   1:  PR[GP1:91,2] = PR[GP1:90,2] + 99.468;
   1:L PR[91] 10mm/sec FINE;
   1:  PR[GP1:91,1] = PR[GP1:90,1] + 74.034;
   1:  PR[GP1:91,2] = PR[GP1:90,2] + 97.039;
   1:L PR[91] 10mm/sec FINE;
   1:  PR[GP1:91,1] = PR[GP1:90,1] + 75.968;
   1:  PR[GP1:91,2] = PR[GP1:90,2] + 94.856;
   1:L PR[91] 10mm/sec FINE;
   1:  PR[GP1:91,1] = PR[GP1:90,1] + 77.516;
   1:  PR[GP1:91,2] = PR[GP1:90,2] + 93.858;
   1:  PR[GP1:91,3] = PR[GP1:90,3] + 42.900;
   1:L PR[91] 10mm/sec FINE;
   1:  PR[GP1:91,1] = PR[GP1:90,1] + 79.283;
   1:  PR[GP1:91,2] = PR[GP1:90,2] + 92.339;
   1:L PR[91] 10mm/sec FINE;
   1:  PR[GP1:91,1] = PR[GP1:90,1] + 81.543;
   1:  PR[GP1:91,2] = PR[GP1:90,2] + 90.798;
   1:L PR[91] 10mm/sec FINE;
   1:  PR[GP1:91,1] = PR[GP1:90,1] + 82.942;
   1:  PR[GP1:91,2] = PR[GP1:90,2] + 89.888;
   1:L PR[91] 10mm/sec FINE;
   1:  PR[GP1:91,1] = PR[GP1:90,1] + 83.980;
   1:  PR[GP1:91,2] = PR[GP1:90,2] + 89.382;
   1:L PR[91] 10mm/sec FINE;
   1:  PR[GP1:91,1] = PR[GP1:90,1] + 87.933;
   1:  PR[GP1:91,2] = PR[GP1:90,2] + 87.648;
   1:L PR[91] 10mm/sec FINE;
   1:  PR[GP1:91,1] = PR[GP1:90,1] + 88.187;
   1:  PR[GP1:91,2] = PR[GP1:90,2] + 87.560;
   1:L PR[91] 10mm/sec FINE;
   1:  PR[GP1:91,1] = PR[GP1:90,1] + 89.431;
   1:  PR[GP1:91,2] = PR[GP1:90,2] + 87.262;
   1:L PR[91] 10mm/sec FINE;
   1:  PR[GP1:91,1] = PR[GP1:90,1] + 92.833;
   1:  PR[GP1:91,2] = PR[GP1:90,2] + 86.250;
   1:L PR[91] 10mm/sec FINE;
   1:  PR[GP1:91,1] = PR[GP1:90,1] + 93.950;
   1:  PR[GP1:91,2] = PR[GP1:90,2] + 85.987;
   1:L PR[91] 10mm/sec FINE;
   1:  PR[GP1:91,1] = PR[GP1:90,1] + 97.467;
   1:  PR[GP1:91,2] = PR[GP1:90,2] + 85.608;
   1:L PR[91] 10mm/sec FINE;
   1:  PR[GP1:91,1] = PR[GP1:90,1] + 100.046;
   1:  PR[GP1:91,2] = PR[GP1:90,2] + 85.501;
   1:L PR[91] 10mm/sec FINE;
   1:  PR[GP1:91,1] = PR[GP1:90,1] + 101.809;
   1:  PR[GP1:91,2] = PR[GP1:90,2] + 85.697;
   1:L PR[91] 10mm/sec FINE;
   1:  PR[GP1:91,1] = PR[GP1:90,1] + 102.507;
   1:  PR[GP1:91,2] = PR[GP1:90,2] + 85.656;
   1:L PR[91] 10mm/sec FINE;
   1:  PR[GP1:91,1] = PR[GP1:90,1] + 104.081;
   1:  PR[GP1:91,2] = PR[GP1:90,2] + 85.414;
   1:L PR[91] 10mm/sec FINE;
   1:  PR[GP1:91,1] = PR[GP1:90,1] + 105.629;
   1:  PR[GP1:91,2] = PR[GP1:90,2] + 85.297;
   1:L PR[91] 10mm/sec FINE;
   1:  PR[GP1:91,1] = PR[GP1:90,1] + 106.776;
   1:L PR[91] 10mm/sec FINE;
   1:  PR[GP1:91,1] = PR[GP1:90,1] + 108.676;
   1:  PR[GP1:91,2] = PR[GP1:90,2] + 85.462;
   1:L PR[91] 10mm/sec FINE;
   1:  PR[GP1:91,1] = PR[GP1:90,1] + 109.474;
   1:  PR[GP1:91,2] = PR[GP1:90,2] + 85.591;
   1:L PR[91] 10mm/sec FINE;
   1:  PR[GP1:91,1] = PR[GP1:90,1] + 111.613;
   1:  PR[GP1:91,2] = PR[GP1:90,2] + 86.140;
   1:L PR[91] 10mm/sec FINE;
   1:  PR[GP1:91,1] = PR[GP1:90,1] + 112.123;
   1:  PR[GP1:91,2] = PR[GP1:90,2] + 86.310;
   1:L PR[91] 10mm/sec FINE;
   1:  PR[GP1:91,1] = PR[GP1:90,1] + 114.339;
   1:  PR[GP1:91,2] = PR[GP1:90,2] + 87.294;
   1:L PR[91] 10mm/sec FINE;
   1:  PR[GP1:91,1] = PR[GP1:90,1] + 114.659;
   1:  PR[GP1:91,2] = PR[GP1:90,2] + 87.463;
   1:L PR[91] 10mm/sec FINE;
   1:  PR[GP1:91,1] = PR[GP1:90,1] + 116.762;
   1:  PR[GP1:91,2] = PR[GP1:90,2] + 88.857;
   1:L PR[91] 10mm/sec FINE;
   1:  PR[GP1:91,1] = PR[GP1:90,1] + 117.014;
   1:  PR[GP1:91,2] = PR[GP1:90,2] + 89.048;
   1:L PR[91] 10mm/sec FINE;
   1:  PR[GP1:91,1] = PR[GP1:90,1] + 118.819;
   1:  PR[GP1:91,2] = PR[GP1:90,2] + 90.739;
   1:L PR[91] 10mm/sec FINE;
   1:  PR[GP1:91,1] = PR[GP1:90,1] + 119.110;
   1:  PR[GP1:91,2] = PR[GP1:90,2] + 91.046;
   1:L PR[91] 10mm/sec FINE;
   1:  PR[GP1:91,1] = PR[GP1:90,1] + 120.475;
   1:  PR[GP1:91,2] = PR[GP1:90,2] + 92.841;
   1:L PR[91] 10mm/sec FINE;
   1:  PR[GP1:91,1] = PR[GP1:90,1] + 120.865;
   1:  PR[GP1:91,2] = PR[GP1:90,2] + 93.418;
   1:L PR[91] 10mm/sec FINE;
   1:  PR[GP1:91,1] = PR[GP1:90,1] + 121.741;
   1:  PR[GP1:91,2] = PR[GP1:90,2] + 95.070;
   1:L PR[91] 10mm/sec FINE;
   1:  PR[GP1:91,1] = PR[GP1:90,1] + 122.220;
   1:  PR[GP1:91,2] = PR[GP1:90,2] + 96.089;
   1:L PR[91] 10mm/sec FINE;
   1:  PR[GP1:91,1] = PR[GP1:90,1] + 122.659;
   1:  PR[GP1:91,2] = PR[GP1:90,2] + 97.354;
   1:L PR[91] 10mm/sec FINE;
   1:  PR[GP1:91,1] = PR[GP1:90,1] + 123.139;
   1:  PR[GP1:91,2] = PR[GP1:90,2] + 98.958;
   1:L PR[91] 10mm/sec FINE;
   1:  PR[GP1:91,1] = PR[GP1:90,1] + 123.264;
   1:  PR[GP1:91,2] = PR[GP1:90,2] + 99.651;
   1:L PR[91] 10mm/sec FINE;
   1:  PR[GP1:91,1] = PR[GP1:90,1] + 123.588;
   1:  PR[GP1:91,2] = PR[GP1:90,2] + 101.921;
   1:L PR[91] 10mm/sec FINE;
   1:  PR[GP1:91,1] = PR[GP1:90,1] + 123.600;
   1:  PR[GP1:91,2] = PR[GP1:90,2] + 104.888;
   1:L PR[91] 10mm/sec FINE;
   1:  PR[GP1:91,1] = PR[GP1:90,1] + 122.995;
   1:  PR[GP1:91,2] = PR[GP1:90,2] + 108.791;
   1:L PR[91] 10mm/sec FINE;
   1:  PR[GP1:91,1] = PR[GP1:90,1] + 121.765;
   1:  PR[GP1:91,2] = PR[GP1:90,2] + 112.407;
   1:L PR[91] 10mm/sec FINE;
   1:  PR[GP1:91,1] = PR[GP1:90,1] + 120.870;
   1:  PR[GP1:91,2] = PR[GP1:90,2] + 113.981;
   1:L PR[91] 10mm/sec FINE;
   1:  PR[GP1:91,1] = PR[GP1:90,1] + 119.893;
   1:  PR[GP1:91,2] = PR[GP1:90,2] + 115.630;
   1:L PR[91] 10mm/sec FINE;
   1:  PR[GP1:91,1] = PR[GP1:90,1] + 119.147;
   1:  PR[GP1:91,2] = PR[GP1:90,2] + 116.492;
   1:L PR[91] 10mm/sec FINE;
   1:  PR[GP1:91,1] = PR[GP1:90,1] + 117.485;
   1:  PR[GP1:91,2] = PR[GP1:90,2] + 118.360;
   1:L PR[91] 10mm/sec FINE;
   1:  PR[GP1:91,1] = PR[GP1:90,1] + 114.657;
   1:  PR[GP1:91,2] = PR[GP1:90,2] + 120.517;
   1:L PR[91] 10mm/sec FINE;
   1:  PR[GP1:91,1] = PR[GP1:90,1] + 111.519;
   1:  PR[GP1:91,2] = PR[GP1:90,2] + 122.048;
   1:L PR[91] 10mm/sec FINE;
   1:  PR[GP1:91,1] = PR[GP1:90,1] + 110.087;
   1:  PR[GP1:91,2] = PR[GP1:90,2] + 122.431;
   1:L PR[91] 10mm/sec FINE;
   1:  PR[GP1:91,1] = PR[GP1:90,1] + 108.168;
   1:  PR[GP1:91,2] = PR[GP1:90,2] + 122.921;
   1:L PR[91] 10mm/sec FINE;
   1:  PR[GP1:91,1] = PR[GP1:90,1] + 104.699;
   1:  PR[GP1:91,2] = PR[GP1:90,2] + 123.124;
   1:L PR[91] 10mm/sec FINE;
   1:  PR[GP1:91,1] = PR[GP1:90,1] + 103.027;
   1:  PR[GP1:91,2] = PR[GP1:90,2] + 122.912;
   1:L PR[91] 10mm/sec FINE;
   1:  PR[GP1:91,1] = PR[GP1:90,1] + 101.276;
   1:  PR[GP1:91,2] = PR[GP1:90,2] + 122.649;
   1:L PR[91] 10mm/sec FINE;
   1:  PR[GP1:91,1] = PR[GP1:90,1] + 99.074;
   1:  PR[GP1:91,2] = PR[GP1:90,2] + 122.005;
   1:L PR[91] 10mm/sec FINE;
   1:  PR[GP1:91,1] = PR[GP1:90,1] + 97.904;
   1:  PR[GP1:91,2] = PR[GP1:90,2] + 121.902;
   1:L PR[91] 10mm/sec FINE;
   1:  PR[GP1:91,1] = PR[GP1:90,1] + 93.801;
   1:  PR[GP1:91,2] = PR[GP1:90,2] + 122.579;
   1:L PR[91] 10mm/sec FINE;
   1:  PR[GP1:91,1] = PR[GP1:90,1] + 93.286;
   1:  PR[GP1:91,2] = PR[GP1:90,2] + 122.645;
   1:L PR[91] 10mm/sec FINE;
   1:  PR[GP1:91,1] = PR[GP1:90,1] + 89.093;
   1:  PR[GP1:91,2] = PR[GP1:90,2] + 122.677;
   1:L PR[91] 10mm/sec FINE;
   1:  PR[GP1:91,1] = PR[GP1:90,1] + 87.629;
   1:  PR[GP1:91,2] = PR[GP1:90,2] + 122.537;
   1:L PR[91] 10mm/sec FINE;
   1:  PR[GP1:91,1] = PR[GP1:90,1] + 85.652;
   1:  PR[GP1:91,2] = PR[GP1:90,2] + 122.207;
   1:L PR[91] 10mm/sec FINE;
   1:  PR[GP1:91,1] = PR[GP1:90,1] + 83.813;
   1:  PR[GP1:91,2] = PR[GP1:90,2] + 121.808;
   1:L PR[91] 10mm/sec FINE;
   1:  PR[GP1:91,1] = PR[GP1:90,1] + 80.795;
   1:  PR[GP1:91,2] = PR[GP1:90,2] + 120.737;
   1:L PR[91] 10mm/sec FINE;
   1:  PR[GP1:91,1] = PR[GP1:90,1] + 78.461;
   1:  PR[GP1:91,2] = PR[GP1:90,2] + 119.530;
   1:L PR[91] 10mm/sec FINE;
   1:  PR[GP1:91,1] = PR[GP1:90,1] + 77.949;
   1:  PR[GP1:91,2] = PR[GP1:90,2] + 119.170;
   1:L PR[91] 10mm/sec FINE;
   1:  PR[GP1:91,1] = PR[GP1:90,1] + 76.319;
   1:  PR[GP1:91,2] = PR[GP1:90,2] + 117.935;
   1:L PR[91] 10mm/sec FINE;
   1:  PR[GP1:91,1] = PR[GP1:90,1] + 74.935;
   1:  PR[GP1:91,2] = PR[GP1:90,2] + 116.491;
   1:L PR[91] 10mm/sec FINE;
   1:  PR[GP1:91,1] = PR[GP1:90,1] + 74.408;
   1:  PR[GP1:91,2] = PR[GP1:90,2] + 115.908;
   1:L PR[91] 10mm/sec FINE;
   1:  PR[GP1:91,1] = PR[GP1:90,1] + 73.372;
   1:  PR[GP1:91,2] = PR[GP1:90,2] + 114.394;
   1:L PR[91] 10mm/sec FINE;
   1:  PR[GP1:91,1] = PR[GP1:90,1] + 72.842;
   1:  PR[GP1:91,2] = PR[GP1:90,2] + 113.448;
   1:L PR[91] 10mm/sec FINE;
   1:  PR[GP1:91,1] = PR[GP1:90,1] + 72.127;
   1:  PR[GP1:91,2] = PR[GP1:90,2] + 111.928;
   1:L PR[91] 10mm/sec FINE;
   1:  PR[GP1:91,1] = PR[GP1:90,1] + 71.355;
   1:  PR[GP1:91,2] = PR[GP1:90,2] + 109.313;
   1:L PR[91] 10mm/sec FINE;
   1:  PR[GP1:91,1] = PR[GP1:90,1] + 71.204;
   1:  PR[GP1:91,2] = PR[GP1:90,2] + 107.968;
   1:L PR[91] 10mm/sec FINE;
   1:  PR[GP1:91,1] = PR[GP1:90,1] + 71.186;
   1:  PR[GP1:91,2] = PR[GP1:90,2] + 106.809;
   1:L PR[91] 10mm/sec FINE;
   1:  PR[GP1:91,1] = PR[GP1:90,1] + 71.282;
   1:  PR[GP1:91,2] = PR[GP1:90,2] + 105.487;
   1:L PR[91] 10mm/sec FINE;
   1:  PR[GP1:91,1] = PR[GP1:90,1] + 71.483;
   1:  PR[GP1:91,2] = PR[GP1:90,2] + 104.578;
   1:L PR[91] 10mm/sec FINE;
   1:  PR[GP1:91,1] = PR[GP1:90,1] + 72.043;
   1:  PR[GP1:91,2] = PR[GP1:90,2] + 102.143;
   1:L PR[91] 10mm/sec FINE;
   1:  PR[GP1:91,1] = PR[GP1:90,1] + 73.160;
   1:  PR[GP1:91,2] = PR[GP1:90,2] + 99.391;
   1:L PR[91] 10mm/sec FINE;
   1:  PR[GP1:91,1] = PR[GP1:90,1] + 74.854;
   1:  PR[GP1:91,2] = PR[GP1:90,2] + 96.763;
   1:L PR[91] 10mm/sec FINE;
   1:  PR[GP1:91,1] = PR[GP1:90,1] + 76.583;
   1:  PR[GP1:91,2] = PR[GP1:90,2] + 94.811;
   1:L PR[91] 10mm/sec FINE;
   1:  PR[GP1:91,1] = PR[GP1:90,1] + 78.494;
   1:  PR[GP1:91,2] = PR[GP1:90,2] + 93.442;
   1:  PR[GP1:91,3] = PR[GP1:90,3] + 43.900;
   1:L PR[91] 10mm/sec FINE;
   1:  PR[GP1:91,1] = PR[GP1:90,1] + 79.972;
   1:  PR[GP1:91,2] = PR[GP1:90,2] + 92.171;
   1:L PR[91] 10mm/sec FINE;
   1:  PR[GP1:91,1] = PR[GP1:90,1] + 82.774;
   1:  PR[GP1:91,2] = PR[GP1:90,2] + 90.260;
   1:L PR[91] 10mm/sec FINE;
   1:  PR[GP1:91,1] = PR[GP1:90,1] + 83.771;
   1:  PR[GP1:91,2] = PR[GP1:90,2] + 89.611;
   1:L PR[91] 10mm/sec FINE;
   1:  PR[GP1:91,1] = PR[GP1:90,1] + 84.510;
   1:  PR[GP1:91,2] = PR[GP1:90,2] + 89.252;
   1:L PR[91] 10mm/sec FINE;
   1:  PR[GP1:91,1] = PR[GP1:90,1] + 88.374;
   1:  PR[GP1:91,2] = PR[GP1:90,2] + 87.556;
   1:L PR[91] 10mm/sec FINE;
   1:  PR[GP1:91,1] = PR[GP1:90,1] + 88.959;
   1:  PR[GP1:91,2] = PR[GP1:90,2] + 87.272;
   1:L PR[91] 10mm/sec FINE;
   1:  PR[GP1:91,1] = PR[GP1:90,1] + 93.314;
   1:  PR[GP1:91,2] = PR[GP1:90,2] + 85.976;
   1:L PR[91] 10mm/sec FINE;
   1:  PR[GP1:91,1] = PR[GP1:90,1] + 94.968;
   1:  PR[GP1:91,2] = PR[GP1:90,2] + 85.587;
   1:L PR[91] 10mm/sec FINE;
   1:  PR[GP1:91,1] = PR[GP1:90,1] + 97.962;
   1:  PR[GP1:91,2] = PR[GP1:90,2] + 85.265;
   1:L PR[91] 10mm/sec FINE;
   1:  PR[GP1:91,1] = PR[GP1:90,1] + 101.083;
   1:  PR[GP1:91,2] = PR[GP1:90,2] + 85.135;
   1:L PR[91] 10mm/sec FINE;
   1:  PR[GP1:91,1] = PR[GP1:90,1] + 102.373;
   1:  PR[GP1:91,2] = PR[GP1:90,2] + 85.288;
   1:L PR[91] 10mm/sec FINE;
   1:  PR[GP1:91,1] = PR[GP1:90,1] + 103.011;
   1:  PR[GP1:91,2] = PR[GP1:90,2] + 85.251;
   1:L PR[91] 10mm/sec FINE;
   1:  PR[GP1:91,1] = PR[GP1:90,1] + 103.965;
   1:  PR[GP1:91,2] = PR[GP1:90,2] + 85.105;
   1:L PR[91] 10mm/sec FINE;
   1:  PR[GP1:91,1] = PR[GP1:90,1] + 106.183;
   1:  PR[GP1:91,2] = PR[GP1:90,2] + 84.937;
   1:L PR[91] 10mm/sec FINE;
   1:  PR[GP1:91,1] = PR[GP1:90,1] + 106.658;
   1:L PR[91] 10mm/sec FINE;
   1:  PR[GP1:91,1] = PR[GP1:90,1] + 109.269;
   1:  PR[GP1:91,2] = PR[GP1:90,2] + 85.163;
   1:L PR[91] 10mm/sec FINE;
   1:  PR[GP1:91,1] = PR[GP1:90,1] + 112.218;
   1:  PR[GP1:91,2] = PR[GP1:90,2] + 85.893;
   1:L PR[91] 10mm/sec FINE;
   1:  PR[GP1:91,1] = PR[GP1:90,1] + 114.511;
   1:  PR[GP1:91,2] = PR[GP1:90,2] + 86.884;
   1:L PR[91] 10mm/sec FINE;
   1:  PR[GP1:91,1] = PR[GP1:90,1] + 114.905;
   1:  PR[GP1:91,2] = PR[GP1:90,2] + 87.073;
   1:L PR[91] 10mm/sec FINE;
   1:  PR[GP1:91,1] = PR[GP1:90,1] + 116.846;
   1:  PR[GP1:91,2] = PR[GP1:90,2] + 88.351;
   1:L PR[91] 10mm/sec FINE;
   1:  PR[GP1:91,1] = PR[GP1:90,1] + 117.292;
   1:  PR[GP1:91,2] = PR[GP1:90,2] + 88.664;
   1:L PR[91] 10mm/sec FINE;
   1:  PR[GP1:91,1] = PR[GP1:90,1] + 118.984;
   1:  PR[GP1:91,2] = PR[GP1:90,2] + 90.264;
   1:L PR[91] 10mm/sec FINE;
   1:  PR[GP1:91,1] = PR[GP1:90,1] + 119.340;
   1:  PR[GP1:91,2] = PR[GP1:90,2] + 90.616;
   1:L PR[91] 10mm/sec FINE;
   1:  PR[GP1:91,1] = PR[GP1:90,1] + 121.015;
   1:  PR[GP1:91,2] = PR[GP1:90,2] + 92.890;
   1:L PR[91] 10mm/sec FINE;
   1:  PR[GP1:91,1] = PR[GP1:90,1] + 121.733;
   1:  PR[GP1:91,2] = PR[GP1:90,2] + 94.321;
   1:L PR[91] 10mm/sec FINE;
   1:  PR[GP1:91,1] = PR[GP1:90,1] + 122.347;
   1:  PR[GP1:91,2] = PR[GP1:90,2] + 95.497;
   1:L PR[91] 10mm/sec FINE;
   1:  PR[GP1:91,1] = PR[GP1:90,1] + 123.107;
   1:  PR[GP1:91,2] = PR[GP1:90,2] + 97.691;
   1:L PR[91] 10mm/sec FINE;
   1:  PR[GP1:91,1] = PR[GP1:90,1] + 123.315;
   1:  PR[GP1:91,2] = PR[GP1:90,2] + 98.385;
   1:L PR[91] 10mm/sec FINE;
   1:  PR[GP1:91,1] = PR[GP1:90,1] + 123.613;
   1:  PR[GP1:91,2] = PR[GP1:90,2] + 100.032;
   1:L PR[91] 10mm/sec FINE;
   1:  PR[GP1:91,1] = PR[GP1:90,1] + 123.806;
   1:  PR[GP1:91,2] = PR[GP1:90,2] + 101.384;
   1:L PR[91] 10mm/sec FINE;
   1:  PR[GP1:91,1] = PR[GP1:90,1] + 123.774;
   1:  PR[GP1:91,2] = PR[GP1:90,2] + 104.410;
   1:L PR[91] 10mm/sec FINE;
   1:  PR[GP1:91,1] = PR[GP1:90,1] + 123.162;
   1:  PR[GP1:91,2] = PR[GP1:90,2] + 108.349;
   1:L PR[91] 10mm/sec FINE;
   1:  PR[GP1:91,1] = PR[GP1:90,1] + 121.855;
   1:  PR[GP1:91,2] = PR[GP1:90,2] + 112.028;
   1:L PR[91] 10mm/sec FINE;
   1:  PR[GP1:91,1] = PR[GP1:90,1] + 119.970;
   1:  PR[GP1:91,2] = PR[GP1:90,2] + 115.291;
   1:L PR[91] 10mm/sec FINE;
   1:  PR[GP1:91,1] = PR[GP1:90,1] + 118.495;
   1:  PR[GP1:91,2] = PR[GP1:90,2] + 116.996;
   1:L PR[91] 10mm/sec FINE;
   1:  PR[GP1:91,1] = PR[GP1:90,1] + 117.555;
   1:  PR[GP1:91,2] = PR[GP1:90,2] + 118.052;
   1:L PR[91] 10mm/sec FINE;
   1:  PR[GP1:91,1] = PR[GP1:90,1] + 116.103;
   1:  PR[GP1:91,2] = PR[GP1:90,2] + 119.185;
   1:L PR[91] 10mm/sec FINE;
   1:  PR[GP1:91,1] = PR[GP1:90,1] + 114.716;
   1:  PR[GP1:91,2] = PR[GP1:90,2] + 120.236;
   1:L PR[91] 10mm/sec FINE;
   1:  PR[GP1:91,1] = PR[GP1:90,1] + 113.082;
   1:  PR[GP1:91,2] = PR[GP1:90,2] + 121.052;
   1:L PR[91] 10mm/sec FINE;
   1:  PR[GP1:91,1] = PR[GP1:90,1] + 111.558;
   1:  PR[GP1:91,2] = PR[GP1:90,2] + 121.790;
   1:L PR[91] 10mm/sec FINE;
   1:  PR[GP1:91,1] = PR[GP1:90,1] + 108.163;
   1:  PR[GP1:91,2] = PR[GP1:90,2] + 122.690;
   1:L PR[91] 10mm/sec FINE;
   1:  PR[GP1:91,1] = PR[GP1:90,1] + 104.735;
   1:  PR[GP1:91,2] = PR[GP1:90,2] + 122.895;
   1:L PR[91] 10mm/sec FINE;
   1:  PR[GP1:91,1] = PR[GP1:90,1] + 101.246;
   1:  PR[GP1:91,2] = PR[GP1:90,2] + 122.446;
   1:L PR[91] 10mm/sec FINE;
   1:  PR[GP1:91,1] = PR[GP1:90,1] + 99.328;
   1:  PR[GP1:91,2] = PR[GP1:90,2] + 121.885;
   1:L PR[91] 10mm/sec FINE;
   1:  PR[GP1:91,1] = PR[GP1:90,1] + 98.158;
   1:  PR[GP1:91,2] = PR[GP1:90,2] + 121.795;
   1:L PR[91] 10mm/sec FINE;
   1:  PR[GP1:91,1] = PR[GP1:90,1] + 94.148;
   1:  PR[GP1:91,2] = PR[GP1:90,2] + 122.433;
   1:L PR[91] 10mm/sec FINE;
   1:  PR[GP1:91,1] = PR[GP1:90,1] + 89.784;
   1:  PR[GP1:91,2] = PR[GP1:90,2] + 122.460;
   1:L PR[91] 10mm/sec FINE;
   1:  PR[GP1:91,1] = PR[GP1:90,1] + 88.694;
   1:  PR[GP1:91,2] = PR[GP1:90,2] + 122.355;
   1:L PR[91] 10mm/sec FINE;
   1:  PR[GP1:91,1] = PR[GP1:90,1] + 86.205;
   1:  PR[GP1:91,2] = PR[GP1:90,2] + 121.940;
   1:L PR[91] 10mm/sec FINE;
   1:  PR[GP1:91,1] = PR[GP1:90,1] + 84.674;
   1:  PR[GP1:91,2] = PR[GP1:90,2] + 121.607;
   1:L PR[91] 10mm/sec FINE;
   1:  PR[GP1:91,1] = PR[GP1:90,1] + 82.722;
   1:  PR[GP1:91,2] = PR[GP1:90,2] + 120.922;
   1:L PR[91] 10mm/sec FINE;
   1:  PR[GP1:91,1] = PR[GP1:90,1] + 81.507;
   1:  PR[GP1:91,2] = PR[GP1:90,2] + 120.475;
   1:L PR[91] 10mm/sec FINE;
   1:  PR[GP1:91,1] = PR[GP1:90,1] + 79.471;
   1:  PR[GP1:91,2] = PR[GP1:90,2] + 119.423;
   1:L PR[91] 10mm/sec FINE;
   1:  PR[GP1:91,1] = PR[GP1:90,1] + 78.997;
   1:  PR[GP1:91,2] = PR[GP1:90,2] + 119.127;
   1:L PR[91] 10mm/sec FINE;
   1:  PR[GP1:91,1] = PR[GP1:90,1] + 77.070;
   1:  PR[GP1:91,2] = PR[GP1:90,2] + 117.744;
   1:L PR[91] 10mm/sec FINE;
   1:  PR[GP1:91,1] = PR[GP1:90,1] + 76.212;
   1:  PR[GP1:91,2] = PR[GP1:90,2] + 116.890;
   1:L PR[91] 10mm/sec FINE;
   1:  PR[GP1:91,1] = PR[GP1:90,1] + 75.232;
   1:  PR[GP1:91,2] = PR[GP1:90,2] + 115.858;
   1:L PR[91] 10mm/sec FINE;
   1:  PR[GP1:91,1] = PR[GP1:90,1] + 73.947;
   1:  PR[GP1:91,2] = PR[GP1:90,2] + 113.980;
   1:L PR[91] 10mm/sec FINE;
   1:  PR[GP1:91,1] = PR[GP1:90,1] + 73.710;
   1:  PR[GP1:91,2] = PR[GP1:90,2] + 113.557;
   1:L PR[91] 10mm/sec FINE;
   1:  PR[GP1:91,1] = PR[GP1:90,1] + 72.804;
   1:  PR[GP1:91,2] = PR[GP1:90,2] + 111.631;
   1:L PR[91] 10mm/sec FINE;
   1:  PR[GP1:91,1] = PR[GP1:90,1] + 72.087;
   1:  PR[GP1:91,2] = PR[GP1:90,2] + 109.185;
   1:L PR[91] 10mm/sec FINE;
   1:  PR[GP1:91,1] = PR[GP1:90,1] + 71.896;
   1:  PR[GP1:91,2] = PR[GP1:90,2] + 107.474;
   1:L PR[91] 10mm/sec FINE;
   1:  PR[GP1:91,1] = PR[GP1:90,1] + 71.886;
   1:  PR[GP1:91,2] = PR[GP1:90,2] + 106.903;
   1:L PR[91] 10mm/sec FINE;
   1:  PR[GP1:91,1] = PR[GP1:90,1] + 72.006;
   1:  PR[GP1:91,2] = PR[GP1:90,2] + 105.257;
   1:L PR[91] 10mm/sec FINE;
   1:  PR[GP1:91,1] = PR[GP1:90,1] + 72.086;
   1:  PR[GP1:91,2] = PR[GP1:90,2] + 104.899;
   1:L PR[91] 10mm/sec FINE;
   1:  PR[GP1:91,1] = PR[GP1:90,1] + 72.779;
   1:  PR[GP1:91,2] = PR[GP1:90,2] + 101.935;
   1:L PR[91] 10mm/sec FINE;
   1:  PR[GP1:91,1] = PR[GP1:90,1] + 73.904;
   1:  PR[GP1:91,2] = PR[GP1:90,2] + 99.261;
   1:L PR[91] 10mm/sec FINE;
   1:  PR[GP1:91,1] = PR[GP1:90,1] + 74.186;
   1:  PR[GP1:91,2] = PR[GP1:90,2] + 98.792;
   1:L PR[91] 10mm/sec FINE;
   1:  PR[GP1:91,1] = PR[GP1:90,1] + 75.674;
   1:  PR[GP1:91,2] = PR[GP1:90,2] + 96.486;
   1:L PR[91] 10mm/sec FINE;
   1:  PR[GP1:91,1] = PR[GP1:90,1] + 77.199;
   1:  PR[GP1:91,2] = PR[GP1:90,2] + 94.765;
   1:L PR[91] 10mm/sec FINE;
   1:  PR[GP1:91,1] = PR[GP1:90,1] + 79.472;
   1:  PR[GP1:91,2] = PR[GP1:90,2] + 93.025;
   1:  PR[GP1:91,3] = PR[GP1:90,3] + 44.900;
   1:L PR[91] 10mm/sec FINE;
   1:  PR[GP1:91,1] = PR[GP1:90,1] + 80.662;
   1:  PR[GP1:91,2] = PR[GP1:90,2] + 92.003;
   1:L PR[91] 10mm/sec FINE;
   1:  PR[GP1:91,1] = PR[GP1:90,1] + 84.006;
   1:  PR[GP1:91,2] = PR[GP1:90,2] + 89.722;
   1:L PR[91] 10mm/sec FINE;
   1:  PR[GP1:91,1] = PR[GP1:90,1] + 84.601;
   1:  PR[GP1:91,2] = PR[GP1:90,2] + 89.334;
   1:L PR[91] 10mm/sec FINE;
   1:  PR[GP1:91,1] = PR[GP1:90,1] + 85.040;
   1:  PR[GP1:91,2] = PR[GP1:90,2] + 89.121;
   1:L PR[91] 10mm/sec FINE;
   1:  PR[GP1:91,1] = PR[GP1:90,1] + 87.368;
   1:  PR[GP1:91,2] = PR[GP1:90,2] + 88.099;
   1:L PR[91] 10mm/sec FINE;
   1:  PR[GP1:91,1] = PR[GP1:90,1] + 89.310;
   1:  PR[GP1:91,2] = PR[GP1:90,2] + 87.124;
   1:L PR[91] 10mm/sec FINE;
   1:  PR[GP1:91,1] = PR[GP1:90,1] + 89.940;
   1:  PR[GP1:91,2] = PR[GP1:90,2] + 86.850;
   1:L PR[91] 10mm/sec FINE;
   1:  PR[GP1:91,1] = PR[GP1:90,1] + 93.796;
   1:  PR[GP1:91,2] = PR[GP1:90,2] + 85.702;
   1:L PR[91] 10mm/sec FINE;
   1:  PR[GP1:91,1] = PR[GP1:90,1] + 95.985;
   1:  PR[GP1:91,2] = PR[GP1:90,2] + 85.188;
   1:L PR[91] 10mm/sec FINE;
   1:  PR[GP1:91,1] = PR[GP1:90,1] + 98.457;
   1:  PR[GP1:91,2] = PR[GP1:90,2] + 84.921;
   1:L PR[91] 10mm/sec FINE;
   1:  PR[GP1:91,1] = PR[GP1:90,1] + 102.120;
   1:  PR[GP1:91,2] = PR[GP1:90,2] + 84.769;
   1:L PR[91] 10mm/sec FINE;
   1:  PR[GP1:91,1] = PR[GP1:90,1] + 102.964;
   1:  PR[GP1:91,2] = PR[GP1:90,2] + 84.876;
   1:L PR[91] 10mm/sec FINE;
   1:  PR[GP1:91,1] = PR[GP1:90,1] + 103.545;
   1:  PR[GP1:91,2] = PR[GP1:90,2] + 84.843;
   1:L PR[91] 10mm/sec FINE;
   1:  PR[GP1:91,1] = PR[GP1:90,1] + 103.849;
   1:  PR[GP1:91,2] = PR[GP1:90,2] + 84.796;
   1:L PR[91] 10mm/sec FINE;
   1:  PR[GP1:91,1] = PR[GP1:90,1] + 106.562;
   1:  PR[GP1:91,2] = PR[GP1:90,2] + 84.578;
   1:L PR[91] 10mm/sec FINE;
   1:  PR[GP1:91,1] = PR[GP1:90,1] + 106.738;
   1:  PR[GP1:91,2] = PR[GP1:90,2] + 84.573;
   1:L PR[91] 10mm/sec FINE;
   1:  PR[GP1:91,1] = PR[GP1:90,1] + 109.227;
   1:  PR[GP1:91,2] = PR[GP1:90,2] + 84.752;
   1:L PR[91] 10mm/sec FINE;
   1:  PR[GP1:91,1] = PR[GP1:90,1] + 109.847;
   1:  PR[GP1:91,2] = PR[GP1:90,2] + 84.831;
   1:L PR[91] 10mm/sec FINE;
   1:  PR[GP1:91,1] = PR[GP1:90,1] + 111.802;
   1:  PR[GP1:91,2] = PR[GP1:90,2] + 85.305;
   1:L PR[91] 10mm/sec FINE;
   1:  PR[GP1:91,1] = PR[GP1:90,1] + 112.757;
   1:  PR[GP1:91,2] = PR[GP1:90,2] + 85.585;
   1:L PR[91] 10mm/sec FINE;
   1:  PR[GP1:91,1] = PR[GP1:90,1] + 114.259;
   1:  PR[GP1:91,2] = PR[GP1:90,2] + 86.234;
   1:L PR[91] 10mm/sec FINE;
   1:  PR[GP1:91,1] = PR[GP1:90,1] + 115.409;
   1:  PR[GP1:91,2] = PR[GP1:90,2] + 86.785;
   1:L PR[91] 10mm/sec FINE;
   1:  PR[GP1:91,1] = PR[GP1:90,1] + 116.568;
   1:  PR[GP1:91,2] = PR[GP1:90,2] + 87.548;
   1:L PR[91] 10mm/sec FINE;
   1:  PR[GP1:91,1] = PR[GP1:90,1] + 117.756;
   1:  PR[GP1:91,2] = PR[GP1:90,2] + 88.382;
   1:L PR[91] 10mm/sec FINE;
   1:  PR[GP1:91,1] = PR[GP1:90,1] + 118.701;
   1:  PR[GP1:91,2] = PR[GP1:90,2] + 89.276;
   1:L PR[91] 10mm/sec FINE;
   1:  PR[GP1:91,1] = PR[GP1:90,1] + 119.764;
   1:  PR[GP1:91,2] = PR[GP1:90,2] + 90.327;
   1:L PR[91] 10mm/sec FINE;
   1:  PR[GP1:91,1] = PR[GP1:90,1] + 121.405;
   1:  PR[GP1:91,2] = PR[GP1:90,2] + 92.581;
   1:L PR[91] 10mm/sec FINE;
   1:  PR[GP1:91,1] = PR[GP1:90,1] + 122.665;
   1:  PR[GP1:91,2] = PR[GP1:90,2] + 95.102;
   1:L PR[91] 10mm/sec FINE;
   1:  PR[GP1:91,1] = PR[GP1:90,1] + 123.530;
   1:  PR[GP1:91,2] = PR[GP1:90,2] + 97.852;
   1:L PR[91] 10mm/sec FINE;
   1:  PR[GP1:91,1] = PR[GP1:90,1] + 123.661;
   1:  PR[GP1:91,2] = PR[GP1:90,2] + 98.750;
   1:L PR[91] 10mm/sec FINE;
   1:  PR[GP1:91,1] = PR[GP1:90,1] + 123.962;
   1:  PR[GP1:91,2] = PR[GP1:90,2] + 100.412;
   1:L PR[91] 10mm/sec FINE;
   1:  PR[GP1:91,1] = PR[GP1:90,1] + 124.024;
   1:  PR[GP1:91,2] = PR[GP1:90,2] + 100.849;
   1:L PR[91] 10mm/sec FINE;
   1:  PR[GP1:91,1] = PR[GP1:90,1] + 123.988;
   1:  PR[GP1:91,2] = PR[GP1:90,2] + 103.924;
   1:L PR[91] 10mm/sec FINE;
   1:  PR[GP1:91,1] = PR[GP1:90,1] + 123.329;
   1:  PR[GP1:91,2] = PR[GP1:90,2] + 107.909;
   1:L PR[91] 10mm/sec FINE;
   1:  PR[GP1:91,1] = PR[GP1:90,1] + 122.045;
   1:  PR[GP1:91,2] = PR[GP1:90,2] + 111.617;
   1:L PR[91] 10mm/sec FINE;
   1:  PR[GP1:91,1] = PR[GP1:90,1] + 121.457;
   1:  PR[GP1:91,2] = PR[GP1:90,2] + 112.647;
   1:L PR[91] 10mm/sec FINE;
   1:  PR[GP1:91,1] = PR[GP1:90,1] + 120.084;
   1:  PR[GP1:91,2] = PR[GP1:90,2] + 114.938;
   1:L PR[91] 10mm/sec FINE;
   1:  PR[GP1:91,1] = PR[GP1:90,1] + 117.626;
   1:  PR[GP1:91,2] = PR[GP1:90,2] + 117.743;
   1:L PR[91] 10mm/sec FINE;
   1:  PR[GP1:91,1] = PR[GP1:90,1] + 114.775;
   1:  PR[GP1:91,2] = PR[GP1:90,2] + 119.954;
   1:L PR[91] 10mm/sec FINE;
   1:  PR[GP1:91,1] = PR[GP1:90,1] + 111.594;
   1:  PR[GP1:91,2] = PR[GP1:90,2] + 121.534;
   1:L PR[91] 10mm/sec FINE;
   1:  PR[GP1:91,1] = PR[GP1:90,1] + 108.197;
   1:  PR[GP1:91,2] = PR[GP1:90,2] + 122.449;
   1:L PR[91] 10mm/sec FINE;
   1:  PR[GP1:91,1] = PR[GP1:90,1] + 104.772;
   1:  PR[GP1:91,2] = PR[GP1:90,2] + 122.665;
   1:L PR[91] 10mm/sec FINE;
   1:  PR[GP1:91,1] = PR[GP1:90,1] + 101.305;
   1:  PR[GP1:91,2] = PR[GP1:90,2] + 122.217;
   1:L PR[91] 10mm/sec FINE;
   1:  PR[GP1:91,1] = PR[GP1:90,1] + 100.761;
   1:  PR[GP1:91,2] = PR[GP1:90,2] + 122.083;
   1:L PR[91] 10mm/sec FINE;
   1:  PR[GP1:91,1] = PR[GP1:90,1] + 99.591;
   1:  PR[GP1:91,2] = PR[GP1:90,2] + 121.748;
   1:L PR[91] 10mm/sec FINE;
   1:  PR[GP1:91,1] = PR[GP1:90,1] + 98.417;
   1:  PR[GP1:91,2] = PR[GP1:90,2] + 121.685;
   1:L PR[91] 10mm/sec FINE;
   1:  PR[GP1:91,1] = PR[GP1:90,1] + 95.476;
   1:  PR[GP1:91,2] = PR[GP1:90,2] + 122.142;
   1:L PR[91] 10mm/sec FINE;
   1:  PR[GP1:91,1] = PR[GP1:90,1] + 94.981;
   1:  PR[GP1:91,2] = PR[GP1:90,2] + 122.206;
   1:L PR[91] 10mm/sec FINE;
   1:  PR[GP1:91,1] = PR[GP1:90,1] + 94.253;
   1:  PR[GP1:91,2] = PR[GP1:90,2] + 122.223;
   1:L PR[91] 10mm/sec FINE;
   1:  PR[GP1:91,1] = PR[GP1:90,1] + 90.474;
   1:  PR[GP1:91,2] = PR[GP1:90,2] + 122.242;
   1:L PR[91] 10mm/sec FINE;
   1:  PR[GP1:91,1] = PR[GP1:90,1] + 89.760;
   1:  PR[GP1:91,2] = PR[GP1:90,2] + 122.173;
   1:L PR[91] 10mm/sec FINE;
   1:  PR[GP1:91,1] = PR[GP1:90,1] + 86.758;
   1:  PR[GP1:91,2] = PR[GP1:90,2] + 121.673;
   1:L PR[91] 10mm/sec FINE;
   1:  PR[GP1:91,1] = PR[GP1:90,1] + 85.535;
   1:  PR[GP1:91,2] = PR[GP1:90,2] + 121.407;
   1:L PR[91] 10mm/sec FINE;
   1:  PR[GP1:91,1] = PR[GP1:90,1] + 83.975;
   1:  PR[GP1:91,2] = PR[GP1:90,2] + 120.859;
   1:L PR[91] 10mm/sec FINE;
   1:  PR[GP1:91,1] = PR[GP1:90,1] + 82.219;
   1:  PR[GP1:91,2] = PR[GP1:90,2] + 120.214;
   1:L PR[91] 10mm/sec FINE;
   1:  PR[GP1:91,1] = PR[GP1:90,1] + 80.485;
   1:  PR[GP1:91,2] = PR[GP1:90,2] + 119.318;
   1:L PR[91] 10mm/sec FINE;
   1:  PR[GP1:91,1] = PR[GP1:90,1] + 79.604;
   1:  PR[GP1:91,2] = PR[GP1:90,2] + 118.768;
   1:L PR[91] 10mm/sec FINE;
   1:  PR[GP1:91,1] = PR[GP1:90,1] + 77.917;
   1:  PR[GP1:91,2] = PR[GP1:90,2] + 117.556;
   1:L PR[91] 10mm/sec FINE;
   1:  PR[GP1:91,1] = PR[GP1:90,1] + 76.002;
   1:  PR[GP1:91,2] = PR[GP1:90,2] + 115.646;
   1:L PR[91] 10mm/sec FINE;
   1:  PR[GP1:91,1] = PR[GP1:90,1] + 74.545;
   1:  PR[GP1:91,2] = PR[GP1:90,2] + 113.567;
   1:L PR[91] 10mm/sec FINE;
   1:  PR[GP1:91,1] = PR[GP1:90,1] + 73.481;
   1:  PR[GP1:91,2] = PR[GP1:90,2] + 111.333;
   1:L PR[91] 10mm/sec FINE;
   1:  PR[GP1:91,1] = PR[GP1:90,1] + 72.819;
   1:  PR[GP1:91,2] = PR[GP1:90,2] + 109.058;
   1:L PR[91] 10mm/sec FINE;
   1:  PR[GP1:91,1] = PR[GP1:90,1] + 72.588;
   1:  PR[GP1:91,2] = PR[GP1:90,2] + 106.990;
   1:L PR[91] 10mm/sec FINE;
   1:  PR[GP1:91,1] = PR[GP1:90,1] + 72.758;
   1:  PR[GP1:91,2] = PR[GP1:90,2] + 105.011;
   1:L PR[91] 10mm/sec FINE;
   1:  PR[GP1:91,1] = PR[GP1:90,1] + 73.497;
   1:  PR[GP1:91,2] = PR[GP1:90,2] + 101.990;
   1:L PR[91] 10mm/sec FINE;
   1:  PR[GP1:91,1] = PR[GP1:90,1] + 73.641;
   1:  PR[GP1:91,2] = PR[GP1:90,2] + 101.525;
   1:L PR[91] 10mm/sec FINE;
   1:  PR[GP1:91,1] = PR[GP1:90,1] + 74.647;
   1:  PR[GP1:91,2] = PR[GP1:90,2] + 99.133;
   1:L PR[91] 10mm/sec FINE;
   1:  PR[GP1:91,1] = PR[GP1:90,1] + 75.205;
   1:  PR[GP1:91,2] = PR[GP1:90,2] + 98.207;
   1:L PR[91] 10mm/sec FINE;
   1:  PR[GP1:91,1] = PR[GP1:90,1] + 76.494;
   1:  PR[GP1:91,2] = PR[GP1:90,2] + 96.210;
   1:L PR[91] 10mm/sec FINE;
   1:  PR[GP1:91,1] = PR[GP1:90,1] + 77.814;
   1:  PR[GP1:91,2] = PR[GP1:90,2] + 94.720;
   1:L PR[91] 10mm/sec FINE;
   1:  PR[GP1:91,1] = PR[GP1:90,1] + 80.451;
   1:  PR[GP1:91,2] = PR[GP1:90,2] + 92.608;
   1:  PR[GP1:91,3] = PR[GP1:90,3] + 45.900;
   1:L PR[91] 10mm/sec FINE;
   1:  PR[GP1:91,1] = PR[GP1:90,1] + 81.351;
   1:  PR[GP1:91,2] = PR[GP1:90,2] + 91.835;
   1:L PR[91] 10mm/sec FINE;
   1:  PR[GP1:91,1] = PR[GP1:90,1] + 85.430;
   1:  PR[GP1:91,2] = PR[GP1:90,2] + 89.059;
   1:L PR[91] 10mm/sec FINE;
   1:  PR[GP1:91,1] = PR[GP1:90,1] + 86.361;
   1:  PR[GP1:91,2] = PR[GP1:90,2] + 88.643;
   1:L PR[91] 10mm/sec FINE;
   1:  PR[GP1:91,1] = PR[GP1:90,1] + 89.797;
   1:  PR[GP1:91,2] = PR[GP1:90,2] + 86.918;
   1:L PR[91] 10mm/sec FINE;
   1:  PR[GP1:91,1] = PR[GP1:90,1] + 90.925;
   1:  PR[GP1:91,2] = PR[GP1:90,2] + 86.426;
   1:L PR[91] 10mm/sec FINE;
   1:  PR[GP1:91,1] = PR[GP1:90,1] + 94.278;
   1:  PR[GP1:91,2] = PR[GP1:90,2] + 85.428;
   1:L PR[91] 10mm/sec FINE;
   1:  PR[GP1:91,1] = PR[GP1:90,1] + 97.002;
   1:  PR[GP1:91,2] = PR[GP1:90,2] + 84.788;
   1:L PR[91] 10mm/sec FINE;
   1:  PR[GP1:91,1] = PR[GP1:90,1] + 98.952;
   1:  PR[GP1:91,2] = PR[GP1:90,2] + 84.578;
   1:L PR[91] 10mm/sec FINE;
   1:  PR[GP1:91,1] = PR[GP1:90,1] + 103.157;
   1:  PR[GP1:91,2] = PR[GP1:90,2] + 84.403;
   1:L PR[91] 10mm/sec FINE;
   1:  PR[GP1:91,1] = PR[GP1:90,1] + 103.581;
   1:  PR[GP1:91,2] = PR[GP1:90,2] + 84.460;
   1:L PR[91] 10mm/sec FINE;
   1:  PR[GP1:91,1] = PR[GP1:90,1] + 104.098;
   1:  PR[GP1:91,2] = PR[GP1:90,2] + 84.432;
   1:L PR[91] 10mm/sec FINE;
   1:  PR[GP1:91,1] = PR[GP1:90,1] + 106.450;
   1:  PR[GP1:91,2] = PR[GP1:90,2] + 84.222;
   1:L PR[91] 10mm/sec FINE;
   1:  PR[GP1:91,1] = PR[GP1:90,1] + 107.345;
   1:  PR[GP1:91,2] = PR[GP1:90,2] + 84.198;
   1:L PR[91] 10mm/sec FINE;
   1:  PR[GP1:91,1] = PR[GP1:90,1] + 109.064;
   1:  PR[GP1:91,2] = PR[GP1:90,2] + 84.321;
   1:L PR[91] 10mm/sec FINE;
   1:  PR[GP1:91,1] = PR[GP1:90,1] + 110.425;
   1:  PR[GP1:91,2] = PR[GP1:90,2] + 84.495;
   1:L PR[91] 10mm/sec FINE;
   1:  PR[GP1:91,1] = PR[GP1:90,1] + 111.590;
   1:  PR[GP1:91,2] = PR[GP1:90,2] + 84.777;
   1:L PR[91] 10mm/sec FINE;
   1:  PR[GP1:91,1] = PR[GP1:90,1] + 113.301;
   1:  PR[GP1:91,2] = PR[GP1:90,2] + 85.278;
   1:L PR[91] 10mm/sec FINE;
   1:  PR[GP1:91,1] = PR[GP1:90,1] + 114.007;
   1:  PR[GP1:91,2] = PR[GP1:90,2] + 85.583;
   1:L PR[91] 10mm/sec FINE;
   1:  PR[GP1:91,1] = PR[GP1:90,1] + 115.914;
   1:  PR[GP1:91,2] = PR[GP1:90,2] + 86.497;
   1:L PR[91] 10mm/sec FINE;
   1:  PR[GP1:91,1] = PR[GP1:90,1] + 116.290;
   1:  PR[GP1:91,2] = PR[GP1:90,2] + 86.745;
   1:L PR[91] 10mm/sec FINE;
   1:  PR[GP1:91,1] = PR[GP1:90,1] + 118.219;
   1:  PR[GP1:91,2] = PR[GP1:90,2] + 88.099;
   1:L PR[91] 10mm/sec FINE;
   1:  PR[GP1:91,1] = PR[GP1:90,1] + 120.189;
   1:  PR[GP1:91,2] = PR[GP1:90,2] + 90.038;
   1:L PR[91] 10mm/sec FINE;
   1:  PR[GP1:91,1] = PR[GP1:90,1] + 121.796;
   1:  PR[GP1:91,2] = PR[GP1:90,2] + 92.272;
   1:L PR[91] 10mm/sec FINE;
   1:  PR[GP1:91,1] = PR[GP1:90,1] + 122.035;
   1:  PR[GP1:91,2] = PR[GP1:90,2] + 92.749;
   1:L PR[91] 10mm/sec FINE;
   1:  PR[GP1:91,1] = PR[GP1:90,1] + 123.031;
   1:  PR[GP1:91,2] = PR[GP1:90,2] + 94.761;
   1:L PR[91] 10mm/sec FINE;
   1:  PR[GP1:91,1] = PR[GP1:90,1] + 123.884;
   1:  PR[GP1:91,2] = PR[GP1:90,2] + 97.469;
   1:L PR[91] 10mm/sec FINE;
   1:  PR[GP1:91,1] = PR[GP1:90,1] + 124.310;
   1:  PR[GP1:91,2] = PR[GP1:90,2] + 100.366;
   1:L PR[91] 10mm/sec FINE;
   1:  PR[GP1:91,1] = PR[GP1:90,1] + 124.265;
   1:  PR[GP1:91,2] = PR[GP1:90,2] + 102.127;
   1:L PR[91] 10mm/sec FINE;
   1:  PR[GP1:91,1] = PR[GP1:90,1] + 124.259;
   1:  PR[GP1:91,2] = PR[GP1:90,2] + 103.436;
   1:L PR[91] 10mm/sec FINE;
   1:  PR[GP1:91,1] = PR[GP1:90,1] + 123.589;
   1:  PR[GP1:91,2] = PR[GP1:90,2] + 107.446;
   1:L PR[91] 10mm/sec FINE;
   1:  PR[GP1:91,1] = PR[GP1:90,1] + 122.701;
   1:  PR[GP1:91,2] = PR[GP1:90,2] + 109.852;
   1:L PR[91] 10mm/sec FINE;
   1:  PR[GP1:91,1] = PR[GP1:90,1] + 122.234;
   1:  PR[GP1:91,2] = PR[GP1:90,2] + 111.206;
   1:L PR[91] 10mm/sec FINE;
   1:  PR[GP1:91,1] = PR[GP1:90,1] + 121.120;
   1:  PR[GP1:91,2] = PR[GP1:90,2] + 113.156;
   1:L PR[91] 10mm/sec FINE;
   1:  PR[GP1:91,1] = PR[GP1:90,1] + 120.280;
   1:  PR[GP1:91,2] = PR[GP1:90,2] + 114.560;
   1:L PR[91] 10mm/sec FINE;
   1:  PR[GP1:91,1] = PR[GP1:90,1] + 119.430;
   1:  PR[GP1:91,2] = PR[GP1:90,2] + 115.550;
   1:L PR[91] 10mm/sec FINE;
   1:  PR[GP1:91,1] = PR[GP1:90,1] + 117.779;
   1:  PR[GP1:91,2] = PR[GP1:90,2] + 117.408;
   1:L PR[91] 10mm/sec FINE;
   1:  PR[GP1:91,1] = PR[GP1:90,1] + 114.868;
   1:  PR[GP1:91,2] = PR[GP1:90,2] + 119.662;
   1:L PR[91] 10mm/sec FINE;
   1:  PR[GP1:91,1] = PR[GP1:90,1] + 111.669;
   1:  PR[GP1:91,2] = PR[GP1:90,2] + 121.266;
   1:L PR[91] 10mm/sec FINE;
   1:  PR[GP1:91,1] = PR[GP1:90,1] + 108.304;
   1:  PR[GP1:91,2] = PR[GP1:90,2] + 122.187;
   1:L PR[91] 10mm/sec FINE;
   1:  PR[GP1:91,1] = PR[GP1:90,1] + 105.889;
   1:  PR[GP1:91,2] = PR[GP1:90,2] + 122.370;
   1:L PR[91] 10mm/sec FINE;
   1:  PR[GP1:91,1] = PR[GP1:90,1] + 104.808;
   1:  PR[GP1:91,2] = PR[GP1:90,2] + 122.436;
   1:L PR[91] 10mm/sec FINE;
   1:  PR[GP1:91,1] = PR[GP1:90,1] + 101.388;
   1:  PR[GP1:91,2] = PR[GP1:90,2] + 121.983;
   1:L PR[91] 10mm/sec FINE;
   1:  PR[GP1:91,1] = PR[GP1:90,1] + 100.770;
   1:  PR[GP1:91,2] = PR[GP1:90,2] + 121.839;
   1:L PR[91] 10mm/sec FINE;
   1:  PR[GP1:91,1] = PR[GP1:90,1] + 99.868;
   1:  PR[GP1:91,2] = PR[GP1:90,2] + 121.598;
   1:L PR[91] 10mm/sec FINE;
   1:  PR[GP1:91,1] = PR[GP1:90,1] + 98.755;
   1:  PR[GP1:91,2] = PR[GP1:90,2] + 121.537;
   1:L PR[91] 10mm/sec FINE;
   1:  PR[GP1:91,1] = PR[GP1:90,1] + 96.676;
   1:  PR[GP1:91,2] = PR[GP1:90,2] + 121.850;
   1:L PR[91] 10mm/sec FINE;
   1:  PR[GP1:91,1] = PR[GP1:90,1] + 95.903;
   1:  PR[GP1:91,2] = PR[GP1:90,2] + 121.943;
   1:L PR[91] 10mm/sec FINE;
   1:  PR[GP1:91,1] = PR[GP1:90,1] + 92.994;
   1:  PR[GP1:91,2] = PR[GP1:90,2] + 122.015;
   1:L PR[91] 10mm/sec FINE;
   1:  PR[GP1:91,1] = PR[GP1:90,1] + 91.164;
   1:  PR[GP1:91,2] = PR[GP1:90,2] + 122.024;
   1:L PR[91] 10mm/sec FINE;
   1:  PR[GP1:91,1] = PR[GP1:90,1] + 90.825;
   1:  PR[GP1:91,2] = PR[GP1:90,2] + 121.991;
   1:L PR[91] 10mm/sec FINE;
   1:  PR[GP1:91,1] = PR[GP1:90,1] + 87.311;
   1:  PR[GP1:91,2] = PR[GP1:90,2] + 121.405;
   1:L PR[91] 10mm/sec FINE;
   1:  PR[GP1:91,1] = PR[GP1:90,1] + 86.396;
   1:  PR[GP1:91,2] = PR[GP1:90,2] + 121.207;
   1:L PR[91] 10mm/sec FINE;
   1:  PR[GP1:91,1] = PR[GP1:90,1] + 85.227;
   1:  PR[GP1:91,2] = PR[GP1:90,2] + 120.796;
   1:L PR[91] 10mm/sec FINE;
   1:  PR[GP1:91,1] = PR[GP1:90,1] + 82.930;
   1:  PR[GP1:91,2] = PR[GP1:90,2] + 119.952;
   1:L PR[91] 10mm/sec FINE;
   1:  PR[GP1:91,1] = PR[GP1:90,1] + 81.500;
   1:  PR[GP1:91,2] = PR[GP1:90,2] + 119.213;
   1:L PR[91] 10mm/sec FINE;
   1:  PR[GP1:91,1] = PR[GP1:90,1] + 80.212;
   1:  PR[GP1:91,2] = PR[GP1:90,2] + 118.408;
   1:L PR[91] 10mm/sec FINE;
   1:  PR[GP1:91,1] = PR[GP1:90,1] + 78.764;
   1:  PR[GP1:91,2] = PR[GP1:90,2] + 117.369;
   1:L PR[91] 10mm/sec FINE;
   1:  PR[GP1:91,1] = PR[GP1:90,1] + 76.744;
   1:  PR[GP1:91,2] = PR[GP1:90,2] + 115.344;
   1:L PR[91] 10mm/sec FINE;
   1:  PR[GP1:91,1] = PR[GP1:90,1] + 75.499;
   1:  PR[GP1:91,2] = PR[GP1:90,2] + 113.578;
   1:L PR[91] 10mm/sec FINE;
   1:  PR[GP1:91,1] = PR[GP1:90,1] + 75.247;
   1:  PR[GP1:91,2] = PR[GP1:90,2] + 113.137;
   1:L PR[91] 10mm/sec FINE;
   1:  PR[GP1:91,1] = PR[GP1:90,1] + 74.294;
   1:  PR[GP1:91,2] = PR[GP1:90,2] + 111.153;
   1:L PR[91] 10mm/sec FINE;
   1:  PR[GP1:91,1] = PR[GP1:90,1] + 73.600;
   1:  PR[GP1:91,2] = PR[GP1:90,2] + 108.762;
   1:L PR[91] 10mm/sec FINE;
   1:  PR[GP1:91,1] = PR[GP1:90,1] + 73.403;
   1:  PR[GP1:91,2] = PR[GP1:90,2] + 106.920;
   1:L PR[91] 10mm/sec FINE;
   1:  PR[GP1:91,1] = PR[GP1:90,1] + 73.551;
   1:  PR[GP1:91,2] = PR[GP1:90,2] + 105.288;
   1:L PR[91] 10mm/sec FINE;
   1:  PR[GP1:91,1] = PR[GP1:90,1] + 73.568;
   1:  PR[GP1:91,2] = PR[GP1:90,2] + 104.713;
   1:L PR[91] 10mm/sec FINE;
   1:  PR[GP1:91,1] = PR[GP1:90,1] + 74.229;
   1:  PR[GP1:91,2] = PR[GP1:90,2] + 101.999;
   1:L PR[91] 10mm/sec FINE;
   1:  PR[GP1:91,1] = PR[GP1:90,1] + 74.506;
   1:  PR[GP1:91,2] = PR[GP1:90,2] + 101.109;
   1:L PR[91] 10mm/sec FINE;
   1:  PR[GP1:91,1] = PR[GP1:90,1] + 75.391;
   1:  PR[GP1:91,2] = PR[GP1:90,2] + 99.004;
   1:L PR[91] 10mm/sec FINE;
   1:  PR[GP1:91,1] = PR[GP1:90,1] + 76.225;
   1:  PR[GP1:91,2] = PR[GP1:90,2] + 97.621;
   1:L PR[91] 10mm/sec FINE;
   1:  PR[GP1:91,1] = PR[GP1:90,1] + 77.314;
   1:  PR[GP1:91,2] = PR[GP1:90,2] + 95.933;
   1:L PR[91] 10mm/sec FINE;
   1:  PR[GP1:91,1] = PR[GP1:90,1] + 78.429;
   1:  PR[GP1:91,2] = PR[GP1:90,2] + 94.674;
   1:L PR[91] 10mm/sec FINE;
   1:  PR[GP1:91,1] = PR[GP1:90,1] + 81.429;
   1:  PR[GP1:91,2] = PR[GP1:90,2] + 92.191;
   1:  PR[GP1:91,3] = PR[GP1:90,3] + 46.900;
   1:L PR[91] 10mm/sec FINE;
   1:  PR[GP1:91,1] = PR[GP1:90,1] + 82.040;
   1:  PR[GP1:91,2] = PR[GP1:90,2] + 91.666;
   1:L PR[91] 10mm/sec FINE;
   1:  PR[GP1:91,1] = PR[GP1:90,1] + 85.444;
   1:  PR[GP1:91,2] = PR[GP1:90,2] + 89.345;
   1:L PR[91] 10mm/sec FINE;
   1:  PR[GP1:91,1] = PR[GP1:90,1] + 86.123;
   1:  PR[GP1:91,2] = PR[GP1:90,2] + 88.834;
   1:L PR[91] 10mm/sec FINE;
   1:  PR[GP1:91,1] = PR[GP1:90,1] + 86.320;
   1:  PR[GP1:91,2] = PR[GP1:90,2] + 88.702;
   1:L PR[91] 10mm/sec FINE;
   1:  PR[GP1:91,1] = PR[GP1:90,1] + 90.285;
   1:  PR[GP1:91,2] = PR[GP1:90,2] + 86.711;
   1:L PR[91] 10mm/sec FINE;
   1:  PR[GP1:91,1] = PR[GP1:90,1] + 91.910;
   1:  PR[GP1:91,2] = PR[GP1:90,2] + 86.002;
   1:L PR[91] 10mm/sec FINE;
   1:  PR[GP1:91,1] = PR[GP1:90,1] + 94.760;
   1:  PR[GP1:91,2] = PR[GP1:90,2] + 85.154;
   1:L PR[91] 10mm/sec FINE;
   1:  PR[GP1:91,1] = PR[GP1:90,1] + 98.019;
   1:  PR[GP1:91,2] = PR[GP1:90,2] + 84.388;
   1:L PR[91] 10mm/sec FINE;
   1:  PR[GP1:91,1] = PR[GP1:90,1] + 99.447;
   1:  PR[GP1:91,2] = PR[GP1:90,2] + 84.234;
   1:L PR[91] 10mm/sec FINE;
   1:  PR[GP1:91,1] = PR[GP1:90,1] + 104.241;
   1:  PR[GP1:91,2] = PR[GP1:90,2] + 84.040;
   1:L PR[91] 10mm/sec FINE;
   1:  PR[GP1:91,1] = PR[GP1:90,1] + 104.698;
   1:  PR[GP1:91,2] = PR[GP1:90,2] + 84.014;
   1:L PR[91] 10mm/sec FINE;
   1:  PR[GP1:91,1] = PR[GP1:90,1] + 106.338;
   1:  PR[GP1:91,2] = PR[GP1:90,2] + 83.866;
   1:L PR[91] 10mm/sec FINE;
   1:  PR[GP1:91,1] = PR[GP1:90,1] + 107.952;
   1:  PR[GP1:91,2] = PR[GP1:90,2] + 83.822;
   1:L PR[91] 10mm/sec FINE;
   1:  PR[GP1:91,1] = PR[GP1:90,1] + 108.900;
   1:  PR[GP1:91,2] = PR[GP1:90,2] + 83.890;
   1:L PR[91] 10mm/sec FINE;
   1:  PR[GP1:91,1] = PR[GP1:90,1] + 111.004;
   1:  PR[GP1:91,2] = PR[GP1:90,2] + 84.158;
   1:L PR[91] 10mm/sec FINE;
   1:  PR[GP1:91,1] = PR[GP1:90,1] + 111.379;
   1:  PR[GP1:91,2] = PR[GP1:90,2] + 84.249;
   1:L PR[91] 10mm/sec FINE;
   1:  PR[GP1:91,1] = PR[GP1:90,1] + 113.788;
   1:  PR[GP1:91,2] = PR[GP1:90,2] + 84.947;
   1:L PR[91] 10mm/sec FINE;
   1:  PR[GP1:91,1] = PR[GP1:90,1] + 116.180;
   1:  PR[GP1:91,2] = PR[GP1:90,2] + 86.039;
   1:L PR[91] 10mm/sec FINE;
   1:  PR[GP1:91,1] = PR[GP1:90,1] + 116.683;
   1:  PR[GP1:91,2] = PR[GP1:90,2] + 86.335;
   1:L PR[91] 10mm/sec FINE;
   1:  PR[GP1:91,1] = PR[GP1:90,1] + 118.421;
   1:  PR[GP1:91,2] = PR[GP1:90,2] + 87.531;
   1:L PR[91] 10mm/sec FINE;
   1:  PR[GP1:91,1] = PR[GP1:90,1] + 119.082;
   1:  PR[GP1:91,2] = PR[GP1:90,2] + 88.103;
   1:L PR[91] 10mm/sec FINE;
   1:  PR[GP1:91,1] = PR[GP1:90,1] + 120.434;
   1:  PR[GP1:91,2] = PR[GP1:90,2] + 89.437;
   1:L PR[91] 10mm/sec FINE;
   1:  PR[GP1:91,1] = PR[GP1:90,1] + 121.003;
   1:  PR[GP1:91,2] = PR[GP1:90,2] + 90.153;
   1:L PR[91] 10mm/sec FINE;
   1:  PR[GP1:91,1] = PR[GP1:90,1] + 122.119;
   1:  PR[GP1:91,2] = PR[GP1:90,2] + 91.735;
   1:L PR[91] 10mm/sec FINE;
   1:  PR[GP1:91,1] = PR[GP1:90,1] + 122.446;
   1:  PR[GP1:91,2] = PR[GP1:90,2] + 92.349;
   1:L PR[91] 10mm/sec FINE;
   1:  PR[GP1:91,1] = PR[GP1:90,1] + 123.395;
   1:  PR[GP1:91,2] = PR[GP1:90,2] + 94.348;
   1:L PR[91] 10mm/sec FINE;
   1:  PR[GP1:91,1] = PR[GP1:90,1] + 123.473;
   1:  PR[GP1:91,2] = PR[GP1:90,2] + 94.583;
   1:L PR[91] 10mm/sec FINE;
   1:  PR[GP1:91,1] = PR[GP1:90,1] + 123.746;
   1:  PR[GP1:91,2] = PR[GP1:90,2] + 95.524;
   1:L PR[91] 10mm/sec FINE;
   1:  PR[GP1:91,1] = PR[GP1:90,1] + 124.238;
   1:  PR[GP1:91,2] = PR[GP1:90,2] + 97.087;
   1:L PR[91] 10mm/sec FINE;
   1:  PR[GP1:91,1] = PR[GP1:90,1] + 124.665;
   1:  PR[GP1:91,2] = PR[GP1:90,2] + 99.937;
   1:L PR[91] 10mm/sec FINE;
   1:  PR[GP1:91,1] = PR[GP1:90,1] + 124.617;
   1:  PR[GP1:91,2] = PR[GP1:90,2] + 101.796;
   1:L PR[91] 10mm/sec FINE;
   1:  PR[GP1:91,1] = PR[GP1:90,1] + 124.569;
   1:  PR[GP1:91,2] = PR[GP1:90,2] + 102.946;
   1:L PR[91] 10mm/sec FINE;
   1:  PR[GP1:91,1] = PR[GP1:90,1] + 124.231;
   1:  PR[GP1:91,2] = PR[GP1:90,2] + 104.809;
   1:L PR[91] 10mm/sec FINE;
   1:  PR[GP1:91,1] = PR[GP1:90,1] + 123.869;
   1:  PR[GP1:91,2] = PR[GP1:90,2] + 106.981;
   1:L PR[91] 10mm/sec FINE;
   1:  PR[GP1:91,1] = PR[GP1:90,1] + 122.486;
   1:  PR[GP1:91,2] = PR[GP1:90,2] + 110.775;
   1:L PR[91] 10mm/sec FINE;
   1:  PR[GP1:91,1] = PR[GP1:90,1] + 121.515;
   1:  PR[GP1:91,2] = PR[GP1:90,2] + 112.385;
   1:L PR[91] 10mm/sec FINE;
   1:  PR[GP1:91,1] = PR[GP1:90,1] + 120.475;
   1:  PR[GP1:91,2] = PR[GP1:90,2] + 114.182;
   1:L PR[91] 10mm/sec FINE;
   1:  PR[GP1:91,1] = PR[GP1:90,1] + 118.963;
   1:  PR[GP1:91,2] = PR[GP1:90,2] + 115.942;
   1:L PR[91] 10mm/sec FINE;
   1:  PR[GP1:91,1] = PR[GP1:90,1] + 117.969;
   1:  PR[GP1:91,2] = PR[GP1:90,2] + 117.061;
   1:L PR[91] 10mm/sec FINE;
   1:  PR[GP1:91,1] = PR[GP1:90,1] + 116.714;
   1:  PR[GP1:91,2] = PR[GP1:90,2] + 118.060;
   1:L PR[91] 10mm/sec FINE;
   1:  PR[GP1:91,1] = PR[GP1:90,1] + 115.045;
   1:  PR[GP1:91,2] = PR[GP1:90,2] + 119.344;
   1:L PR[91] 10mm/sec FINE;
   1:  PR[GP1:91,1] = PR[GP1:90,1] + 113.948;
   1:  PR[GP1:91,2] = PR[GP1:90,2] + 119.913;
   1:L PR[91] 10mm/sec FINE;
   1:  PR[GP1:91,1] = PR[GP1:90,1] + 111.823;
   1:  PR[GP1:91,2] = PR[GP1:90,2] + 120.975;
   1:L PR[91] 10mm/sec FINE;
   1:  PR[GP1:91,1] = PR[GP1:90,1] + 110.307;
   1:  PR[GP1:91,2] = PR[GP1:90,2] + 121.410;
   1:L PR[91] 10mm/sec FINE;
   1:  PR[GP1:91,1] = PR[GP1:90,1] + 108.412;
   1:  PR[GP1:91,2] = PR[GP1:90,2] + 121.926;
   1:L PR[91] 10mm/sec FINE;
   1:  PR[GP1:91,1] = PR[GP1:90,1] + 104.884;
   1:  PR[GP1:91,2] = PR[GP1:90,2] + 122.194;
   1:L PR[91] 10mm/sec FINE;
   1:  PR[GP1:91,1] = PR[GP1:90,1] + 104.342;
   1:  PR[GP1:91,2] = PR[GP1:90,2] + 122.135;
   1:L PR[91] 10mm/sec FINE;
   1:  PR[GP1:91,1] = PR[GP1:90,1] + 101.473;
   1:  PR[GP1:91,2] = PR[GP1:90,2] + 121.750;
   1:L PR[91] 10mm/sec FINE;
   1:  PR[GP1:91,1] = PR[GP1:90,1] + 100.157;
   1:  PR[GP1:91,2] = PR[GP1:90,2] + 121.433;
   1:L PR[91] 10mm/sec FINE;
   1:  PR[GP1:91,1] = PR[GP1:90,1] + 99.102;
   1:  PR[GP1:91,2] = PR[GP1:90,2] + 121.378;
   1:L PR[91] 10mm/sec FINE;
   1:  PR[GP1:91,1] = PR[GP1:90,1] + 97.412;
   1:  PR[GP1:91,2] = PR[GP1:90,2] + 121.615;
   1:L PR[91] 10mm/sec FINE;
   1:  PR[GP1:91,1] = PR[GP1:90,1] + 96.608;
   1:  PR[GP1:91,2] = PR[GP1:90,2] + 121.694;
   1:L PR[91] 10mm/sec FINE;
   1:  PR[GP1:91,1] = PR[GP1:90,1] + 95.564;
   1:  PR[GP1:91,2] = PR[GP1:90,2] + 121.699;
   1:L PR[91] 10mm/sec FINE;
   1:  PR[GP1:91,1] = PR[GP1:90,1] + 91.862;
   1:  PR[GP1:91,2] = PR[GP1:90,2] + 121.803;
   1:L PR[91] 10mm/sec FINE;
   1:  PR[GP1:91,1] = PR[GP1:90,1] + 87.864;
   1:  PR[GP1:91,2] = PR[GP1:90,2] + 121.138;
   1:L PR[91] 10mm/sec FINE;
   1:  PR[GP1:91,1] = PR[GP1:90,1] + 87.259;
   1:  PR[GP1:91,2] = PR[GP1:90,2] + 121.007;
   1:L PR[91] 10mm/sec FINE;
   1:  PR[GP1:91,1] = PR[GP1:90,1] + 83.641;
   1:  PR[GP1:91,2] = PR[GP1:90,2] + 119.690;
   1:L PR[91] 10mm/sec FINE;
   1:  PR[GP1:91,1] = PR[GP1:90,1] + 82.514;
   1:  PR[GP1:91,2] = PR[GP1:90,2] + 119.108;
   1:L PR[91] 10mm/sec FINE;
   1:  PR[GP1:91,1] = PR[GP1:90,1] + 80.819;
   1:  PR[GP1:91,2] = PR[GP1:90,2] + 118.049;
   1:L PR[91] 10mm/sec FINE;
   1:  PR[GP1:91,1] = PR[GP1:90,1] + 79.611;
   1:  PR[GP1:91,2] = PR[GP1:90,2] + 117.181;
   1:L PR[91] 10mm/sec FINE;
   1:  PR[GP1:91,1] = PR[GP1:90,1] + 78.387;
   1:  PR[GP1:91,2] = PR[GP1:90,2] + 115.964;
   1:L PR[91] 10mm/sec FINE;
   1:  PR[GP1:91,1] = PR[GP1:90,1] + 77.487;
   1:  PR[GP1:91,2] = PR[GP1:90,2] + 115.044;
   1:L PR[91] 10mm/sec FINE;
   1:  PR[GP1:91,1] = PR[GP1:90,1] + 76.421;
   1:  PR[GP1:91,2] = PR[GP1:90,2] + 113.532;
   1:L PR[91] 10mm/sec FINE;
   1:  PR[GP1:91,1] = PR[GP1:90,1] + 75.945;
   1:  PR[GP1:91,2] = PR[GP1:90,2] + 112.699;
   1:L PR[91] 10mm/sec FINE;
   1:  PR[GP1:91,1] = PR[GP1:90,1] + 75.122;
   1:  PR[GP1:91,2] = PR[GP1:90,2] + 110.986;
   1:L PR[91] 10mm/sec FINE;
   1:  PR[GP1:91,1] = PR[GP1:90,1] + 74.388;
   1:  PR[GP1:91,2] = PR[GP1:90,2] + 108.436;
   1:L PR[91] 10mm/sec FINE;
   1:  PR[GP1:91,1] = PR[GP1:90,1] + 74.219;
   1:  PR[GP1:91,2] = PR[GP1:90,2] + 106.850;
   1:L PR[91] 10mm/sec FINE;
   1:  PR[GP1:91,1] = PR[GP1:90,1] + 74.346;
   1:  PR[GP1:91,2] = PR[GP1:90,2] + 105.443;
   1:L PR[91] 10mm/sec FINE;
   1:  PR[GP1:91,1] = PR[GP1:90,1] + 74.378;
   1:  PR[GP1:91,2] = PR[GP1:90,2] + 104.421;
   1:L PR[91] 10mm/sec FINE;
   1:  PR[GP1:91,1] = PR[GP1:90,1] + 74.961;
   1:  PR[GP1:91,2] = PR[GP1:90,2] + 102.008;
   1:L PR[91] 10mm/sec FINE;
   1:  PR[GP1:91,1] = PR[GP1:90,1] + 75.371;
   1:  PR[GP1:91,2] = PR[GP1:90,2] + 100.693;
   1:L PR[91] 10mm/sec FINE;
   1:  PR[GP1:91,1] = PR[GP1:90,1] + 76.135;
   1:  PR[GP1:91,2] = PR[GP1:90,2] + 98.876;
   1:L PR[91] 10mm/sec FINE;
   1:  PR[GP1:91,1] = PR[GP1:90,1] + 77.244;
   1:  PR[GP1:91,2] = PR[GP1:90,2] + 97.036;
   1:L PR[91] 10mm/sec FINE;
   1:  PR[GP1:91,1] = PR[GP1:90,1] + 78.134;
   1:  PR[GP1:91,2] = PR[GP1:90,2] + 95.657;
   1:L PR[91] 10mm/sec FINE;
   1:  PR[GP1:91,1] = PR[GP1:90,1] + 79.044;
   1:  PR[GP1:91,2] = PR[GP1:90,2] + 94.629;
   1:L PR[91] 10mm/sec FINE;
   1:  PR[GP1:91,1] = PR[GP1:90,1] + 82.408;
   1:  PR[GP1:91,2] = PR[GP1:90,2] + 91.775;
   1:  PR[GP1:91,3] = PR[GP1:90,3] + 47.900;
   1:L PR[91] 10mm/sec FINE;
   1:  PR[GP1:91,1] = PR[GP1:90,1] + 82.730;
   1:  PR[GP1:91,2] = PR[GP1:90,2] + 91.498;
   1:L PR[91] 10mm/sec FINE;
   1:  PR[GP1:91,1] = PR[GP1:90,1] + 84.559;
   1:  PR[GP1:91,2] = PR[GP1:90,2] + 90.251;
   1:L PR[91] 10mm/sec FINE;
   1:  PR[GP1:91,1] = PR[GP1:90,1] + 86.634;
   1:  PR[GP1:91,2] = PR[GP1:90,2] + 88.690;
   1:L PR[91] 10mm/sec FINE;
   1:  PR[GP1:91,1] = PR[GP1:90,1] + 87.265;
   1:  PR[GP1:91,2] = PR[GP1:90,2] + 88.265;
   1:L PR[91] 10mm/sec FINE;
   1:  PR[GP1:91,1] = PR[GP1:90,1] + 90.772;
   1:  PR[GP1:91,2] = PR[GP1:90,2] + 86.504;
   1:L PR[91] 10mm/sec FINE;
   1:  PR[GP1:91,1] = PR[GP1:90,1] + 92.895;
   1:  PR[GP1:91,2] = PR[GP1:90,2] + 85.578;
   1:L PR[91] 10mm/sec FINE;
   1:  PR[GP1:91,1] = PR[GP1:90,1] + 95.241;
   1:  PR[GP1:91,2] = PR[GP1:90,2] + 84.880;
   1:L PR[91] 10mm/sec FINE;
   1:  PR[GP1:91,1] = PR[GP1:90,1] + 99.036;
   1:  PR[GP1:91,2] = PR[GP1:90,2] + 83.988;
   1:L PR[91] 10mm/sec FINE;
   1:  PR[GP1:91,1] = PR[GP1:90,1] + 99.942;
   1:  PR[GP1:91,2] = PR[GP1:90,2] + 83.891;
   1:L PR[91] 10mm/sec FINE;
   1:  PR[GP1:91,1] = PR[GP1:90,1] + 103.095;
   1:  PR[GP1:91,2] = PR[GP1:90,2] + 83.760;
   1:L PR[91] 10mm/sec FINE;
   1:  PR[GP1:91,1] = PR[GP1:90,1] + 104.820;
   1:  PR[GP1:91,2] = PR[GP1:90,2] + 83.594;
   1:L PR[91] 10mm/sec FINE;
   1:  PR[GP1:91,1] = PR[GP1:90,1] + 104.848;
   1:  PR[GP1:91,2] = PR[GP1:90,2] + 83.618;
   1:L PR[91] 10mm/sec FINE;
   1:  PR[GP1:91,1] = PR[GP1:90,1] + 105.332;
   1:  PR[GP1:91,2] = PR[GP1:90,2] + 83.592;
   1:L PR[91] 10mm/sec FINE;
   1:  PR[GP1:91,1] = PR[GP1:90,1] + 106.225;
   1:  PR[GP1:91,2] = PR[GP1:90,2] + 83.510;
   1:L PR[91] 10mm/sec FINE;
   1:  PR[GP1:91,1] = PR[GP1:90,1] + 108.555;
   1:  PR[GP1:91,2] = PR[GP1:90,2] + 83.447;
   1:L PR[91] 10mm/sec FINE;
   1:  PR[GP1:91,1] = PR[GP1:90,1] + 111.254;
   1:  PR[GP1:91,2] = PR[GP1:90,2] + 83.746;
   1:L PR[91] 10mm/sec FINE;
   1:  PR[GP1:91,1] = PR[GP1:90,1] + 111.772;
   1:  PR[GP1:91,2] = PR[GP1:90,2] + 83.843;
   1:L PR[91] 10mm/sec FINE;
   1:  PR[GP1:91,1] = PR[GP1:90,1] + 113.754;
   1:  PR[GP1:91,2] = PR[GP1:90,2] + 84.384;
   1:L PR[91] 10mm/sec FINE;
   1:  PR[GP1:91,1] = PR[GP1:90,1] + 114.910;
   1:  PR[GP1:91,2] = PR[GP1:90,2] + 84.813;
   1:L PR[91] 10mm/sec FINE;
   1:  PR[GP1:91,1] = PR[GP1:90,1] + 116.196;
   1:  PR[GP1:91,2] = PR[GP1:90,2] + 85.404;
   1:L PR[91] 10mm/sec FINE;
   1:  PR[GP1:91,1] = PR[GP1:90,1] + 117.734;
   1:  PR[GP1:91,2] = PR[GP1:90,2] + 86.310;
   1:L PR[91] 10mm/sec FINE;
   1:  PR[GP1:91,1] = PR[GP1:90,1] + 118.512;
   1:  PR[GP1:91,2] = PR[GP1:90,2] + 86.846;
   1:L PR[91] 10mm/sec FINE;
   1:  PR[GP1:91,1] = PR[GP1:90,1] + 120.110;
   1:  PR[GP1:91,2] = PR[GP1:90,2] + 88.229;
   1:L PR[91] 10mm/sec FINE;
   1:  PR[GP1:91,1] = PR[GP1:90,1] + 120.613;
   1:  PR[GP1:91,2] = PR[GP1:90,2] + 88.725;
   1:L PR[91] 10mm/sec FINE;
   1:  PR[GP1:91,1] = PR[GP1:90,1] + 121.962;
   1:  PR[GP1:91,2] = PR[GP1:90,2] + 90.421;
   1:L PR[91] 10mm/sec FINE;
   1:  PR[GP1:91,1] = PR[GP1:90,1] + 122.389;
   1:  PR[GP1:91,2] = PR[GP1:90,2] + 91.027;
   1:L PR[91] 10mm/sec FINE;
   1:  PR[GP1:91,1] = PR[GP1:90,1] + 123.302;
   1:  PR[GP1:91,2] = PR[GP1:90,2] + 92.738;
   1:L PR[91] 10mm/sec FINE;
   1:  PR[GP1:91,1] = PR[GP1:90,1] + 123.749;
   1:  PR[GP1:91,2] = PR[GP1:90,2] + 93.679;
   1:L PR[91] 10mm/sec FINE;
   1:  PR[GP1:91,1] = PR[GP1:90,1] + 124.205;
   1:  PR[GP1:91,2] = PR[GP1:90,2] + 95.062;
   1:L PR[91] 10mm/sec FINE;
   1:  PR[GP1:91,1] = PR[GP1:90,1] + 124.637;
   1:  PR[GP1:91,2] = PR[GP1:90,2] + 96.551;
   1:L PR[91] 10mm/sec FINE;
   1:  PR[GP1:91,1] = PR[GP1:90,1] + 124.753;
   1:  PR[GP1:91,2] = PR[GP1:90,2] + 97.324;
   1:L PR[91] 10mm/sec FINE;
   1:  PR[GP1:91,1] = PR[GP1:90,1] + 125.020;
   1:  PR[GP1:91,2] = PR[GP1:90,2] + 99.504;
   1:L PR[91] 10mm/sec FINE;
   1:  PR[GP1:91,1] = PR[GP1:90,1] + 124.948;
   1:  PR[GP1:91,2] = PR[GP1:90,2] + 102.475;
   1:L PR[91] 10mm/sec FINE;
   1:  PR[GP1:91,1] = PR[GP1:90,1] + 124.178;
   1:  PR[GP1:91,2] = PR[GP1:90,2] + 106.513;
   1:L PR[91] 10mm/sec FINE;
   1:  PR[GP1:91,1] = PR[GP1:90,1] + 123.927;
   1:  PR[GP1:91,2] = PR[GP1:90,2] + 107.161;
   1:L PR[91] 10mm/sec FINE;
   1:  PR[GP1:91,1] = PR[GP1:90,1] + 122.789;
   1:  PR[GP1:91,2] = PR[GP1:90,2] + 110.338;
   1:L PR[91] 10mm/sec FINE;
   1:  PR[GP1:91,1] = PR[GP1:90,1] + 122.041;
   1:  PR[GP1:91,2] = PR[GP1:90,2] + 111.624;
   1:L PR[91] 10mm/sec FINE;
   1:  PR[GP1:91,1] = PR[GP1:90,1] + 120.719;
   1:  PR[GP1:91,2] = PR[GP1:90,2] + 113.787;
   1:L PR[91] 10mm/sec FINE;
   1:  PR[GP1:91,1] = PR[GP1:90,1] + 119.591;
   1:  PR[GP1:91,2] = PR[GP1:90,2] + 115.060;
   1:L PR[91] 10mm/sec FINE;
   1:  PR[GP1:91,1] = PR[GP1:90,1] + 118.158;
   1:  PR[GP1:91,2] = PR[GP1:90,2] + 116.715;
   1:L PR[91] 10mm/sec FINE;
   1:  PR[GP1:91,1] = PR[GP1:90,1] + 116.149;
   1:  PR[GP1:91,2] = PR[GP1:90,2] + 118.313;
   1:L PR[91] 10mm/sec FINE;
   1:  PR[GP1:91,1] = PR[GP1:90,1] + 115.223;
   1:  PR[GP1:91,2] = PR[GP1:90,2] + 119.026;
   1:L PR[91] 10mm/sec FINE;
   1:  PR[GP1:91,1] = PR[GP1:90,1] + 113.258;
   1:  PR[GP1:91,2] = PR[GP1:90,2] + 120.044;
   1:L PR[91] 10mm/sec FINE;
   1:  PR[GP1:91,1] = PR[GP1:90,1] + 111.979;
   1:  PR[GP1:91,2] = PR[GP1:90,2] + 120.684;
   1:L PR[91] 10mm/sec FINE;
   1:  PR[GP1:91,1] = PR[GP1:90,1] + 108.520;
   1:  PR[GP1:91,2] = PR[GP1:90,2] + 121.664;
   1:L PR[91] 10mm/sec FINE;
   1:  PR[GP1:91,1] = PR[GP1:90,1] + 105.039;
   1:  PR[GP1:91,2] = PR[GP1:90,2] + 121.930;
   1:L PR[91] 10mm/sec FINE;
   1:  PR[GP1:91,1] = PR[GP1:90,1] + 102.957;
   1:  PR[GP1:91,2] = PR[GP1:90,2] + 121.704;
   1:L PR[91] 10mm/sec FINE;
   1:  PR[GP1:91,1] = PR[GP1:90,1] + 101.556;
   1:  PR[GP1:91,2] = PR[GP1:90,2] + 121.516;
   1:L PR[91] 10mm/sec FINE;
   1:  PR[GP1:91,1] = PR[GP1:90,1] + 100.460;
   1:  PR[GP1:91,2] = PR[GP1:90,2] + 121.257;
   1:L PR[91] 10mm/sec FINE;
   1:  PR[GP1:91,1] = PR[GP1:90,1] + 99.461;
   1:  PR[GP1:91,2] = PR[GP1:90,2] + 121.206;
   1:L PR[91] 10mm/sec FINE;
   1:  PR[GP1:91,1] = PR[GP1:90,1] + 98.008;
   1:  PR[GP1:91,2] = PR[GP1:90,2] + 121.390;
   1:L PR[91] 10mm/sec FINE;
   1:  PR[GP1:91,1] = PR[GP1:90,1] + 97.415;
   1:  PR[GP1:91,2] = PR[GP1:90,2] + 121.438;
   1:L PR[91] 10mm/sec FINE;
   1:  PR[GP1:91,1] = PR[GP1:90,1] + 95.925;
   1:  PR[GP1:91,2] = PR[GP1:90,2] + 121.445;
   1:L PR[91] 10mm/sec FINE;
   1:  PR[GP1:91,1] = PR[GP1:90,1] + 92.625;
   1:  PR[GP1:91,2] = PR[GP1:90,2] + 121.537;
   1:L PR[91] 10mm/sec FINE;
   1:  PR[GP1:91,1] = PR[GP1:90,1] + 90.383;
   1:  PR[GP1:91,2] = PR[GP1:90,2] + 121.199;
   1:L PR[91] 10mm/sec FINE;
   1:  PR[GP1:91,1] = PR[GP1:90,1] + 88.417;
   1:  PR[GP1:91,2] = PR[GP1:90,2] + 120.871;
   1:L PR[91] 10mm/sec FINE;
   1:  PR[GP1:91,1] = PR[GP1:90,1] + 88.120;
   1:  PR[GP1:91,2] = PR[GP1:90,2] + 120.807;
   1:L PR[91] 10mm/sec FINE;
   1:  PR[GP1:91,1] = PR[GP1:90,1] + 84.352;
   1:  PR[GP1:91,2] = PR[GP1:90,2] + 119.428;
   1:L PR[91] 10mm/sec FINE;
   1:  PR[GP1:91,1] = PR[GP1:90,1] + 83.529;
   1:  PR[GP1:91,2] = PR[GP1:90,2] + 119.003;
   1:L PR[91] 10mm/sec FINE;
   1:  PR[GP1:91,1] = PR[GP1:90,1] + 81.427;
   1:  PR[GP1:91,2] = PR[GP1:90,2] + 117.690;
   1:L PR[91] 10mm/sec FINE;
   1:  PR[GP1:91,1] = PR[GP1:90,1] + 80.458;
   1:  PR[GP1:91,2] = PR[GP1:90,2] + 116.994;
   1:L PR[91] 10mm/sec FINE;
   1:  PR[GP1:91,1] = PR[GP1:90,1] + 79.474;
   1:  PR[GP1:91,2] = PR[GP1:90,2] + 116.016;
   1:L PR[91] 10mm/sec FINE;
   1:  PR[GP1:91,1] = PR[GP1:90,1] + 78.230;
   1:  PR[GP1:91,2] = PR[GP1:90,2] + 114.743;
   1:L PR[91] 10mm/sec FINE;
   1:  PR[GP1:91,1] = PR[GP1:90,1] + 77.343;
   1:  PR[GP1:91,2] = PR[GP1:90,2] + 113.485;
   1:L PR[91] 10mm/sec FINE;
   1:  PR[GP1:91,1] = PR[GP1:90,1] + 76.643;
   1:  PR[GP1:91,2] = PR[GP1:90,2] + 112.261;
   1:L PR[91] 10mm/sec FINE;
   1:  PR[GP1:91,1] = PR[GP1:90,1] + 75.950;
   1:  PR[GP1:91,2] = PR[GP1:90,2] + 110.818;
   1:L PR[91] 10mm/sec FINE;
   1:  PR[GP1:91,1] = PR[GP1:90,1] + 75.516;
   1:  PR[GP1:91,2] = PR[GP1:90,2] + 109.335;
   1:L PR[91] 10mm/sec FINE;
   1:  PR[GP1:91,1] = PR[GP1:90,1] + 75.177;
   1:  PR[GP1:91,2] = PR[GP1:90,2] + 108.111;
   1:L PR[91] 10mm/sec FINE;
   1:  PR[GP1:91,1] = PR[GP1:90,1] + 75.035;
   1:  PR[GP1:91,2] = PR[GP1:90,2] + 106.781;
   1:L PR[91] 10mm/sec FINE;
   1:  PR[GP1:91,1] = PR[GP1:90,1] + 75.142;
   1:  PR[GP1:91,2] = PR[GP1:90,2] + 105.597;
   1:L PR[91] 10mm/sec FINE;
   1:  PR[GP1:91,1] = PR[GP1:90,1] + 75.187;
   1:  PR[GP1:91,2] = PR[GP1:90,2] + 104.129;
   1:L PR[91] 10mm/sec FINE;
   1:  PR[GP1:91,1] = PR[GP1:90,1] + 75.627;
   1:  PR[GP1:91,2] = PR[GP1:90,2] + 102.341;
   1:L PR[91] 10mm/sec FINE;
   1:  PR[GP1:91,1] = PR[GP1:90,1] + 75.694;
   1:  PR[GP1:91,2] = PR[GP1:90,2] + 102.014;
   1:L PR[91] 10mm/sec FINE;
   1:  PR[GP1:91,1] = PR[GP1:90,1] + 76.236;
   1:  PR[GP1:91,2] = PR[GP1:90,2] + 100.276;
   1:L PR[91] 10mm/sec FINE;
   1:  PR[GP1:91,1] = PR[GP1:90,1] + 76.878;
   1:  PR[GP1:91,2] = PR[GP1:90,2] + 98.748;
   1:L PR[91] 10mm/sec FINE;
   1:  PR[GP1:91,1] = PR[GP1:90,1] + 78.263;
   1:  PR[GP1:91,2] = PR[GP1:90,2] + 96.450;
   1:L PR[91] 10mm/sec FINE;
   1:  PR[GP1:91,1] = PR[GP1:90,1] + 78.954;
   1:  PR[GP1:91,2] = PR[GP1:90,2] + 95.380;
   1:L PR[91] 10mm/sec FINE;
   1:  PR[GP1:91,1] = PR[GP1:90,1] + 79.660;
   1:  PR[GP1:91,2] = PR[GP1:90,2] + 94.583;
   1:L PR[91] 10mm/sec FINE;
   1:  PR[GP1:91,1] = PR[GP1:90,1] + 80.275;
   1:  PR[GP1:91,2] = PR[GP1:90,2] + 94.538;
   1:  PR[GP1:91,3] = PR[GP1:90,3] + 48.900;
   1:L PR[91] 10mm/sec FINE;
   1:  PR[GP1:91,1] = PR[GP1:90,1] + 83.382;
   1:  PR[GP1:91,2] = PR[GP1:90,2] + 91.363;
   1:L PR[91] 10mm/sec FINE;
   1:  PR[GP1:91,1] = PR[GP1:90,1] + 87.145;
   1:  PR[GP1:91,2] = PR[GP1:90,2] + 88.546;
   1:L PR[91] 10mm/sec FINE;
   1:  PR[GP1:91,1] = PR[GP1:90,1] + 88.210;
   1:  PR[GP1:91,2] = PR[GP1:90,2] + 87.828;
   1:L PR[91] 10mm/sec FINE;
   1:  PR[GP1:91,1] = PR[GP1:90,1] + 91.259;
   1:  PR[GP1:91,2] = PR[GP1:90,2] + 86.297;
   1:L PR[91] 10mm/sec FINE;
   1:  PR[GP1:91,1] = PR[GP1:90,1] + 93.880;
   1:  PR[GP1:91,2] = PR[GP1:90,2] + 85.155;
   1:L PR[91] 10mm/sec FINE;
   1:  PR[GP1:91,1] = PR[GP1:90,1] + 95.723;
   1:  PR[GP1:91,2] = PR[GP1:90,2] + 84.606;
   1:L PR[91] 10mm/sec FINE;
   1:  PR[GP1:91,1] = PR[GP1:90,1] + 100.053;
   1:  PR[GP1:91,2] = PR[GP1:90,2] + 83.589;
   1:L PR[91] 10mm/sec FINE;
   1:  PR[GP1:91,1] = PR[GP1:90,1] + 100.437;
   1:  PR[GP1:91,2] = PR[GP1:90,2] + 83.547;
   1:L PR[91] 10mm/sec FINE;
   1:  PR[GP1:91,1] = PR[GP1:90,1] + 101.810;
   1:  PR[GP1:91,2] = PR[GP1:90,2] + 83.490;
   1:L PR[91] 10mm/sec FINE;
   1:  PR[GP1:91,1] = PR[GP1:90,1] + 105.488;
   1:  PR[GP1:91,2] = PR[GP1:90,2] + 83.136;
   1:L PR[91] 10mm/sec FINE;
   1:  PR[GP1:91,1] = PR[GP1:90,1] + 105.603;
   1:  PR[GP1:91,2] = PR[GP1:90,2] + 83.184;
   1:L PR[91] 10mm/sec FINE;
   1:  PR[GP1:91,1] = PR[GP1:90,1] + 108.634;
   1:  PR[GP1:91,2] = PR[GP1:90,2] + 83.049;
   1:L PR[91] 10mm/sec FINE;
   1:  PR[GP1:91,1] = PR[GP1:90,1] + 109.368;
   1:  PR[GP1:91,2] = PR[GP1:90,2] + 83.065;
   1:L PR[91] 10mm/sec FINE;
   1:  PR[GP1:91,1] = PR[GP1:90,1] + 111.171;
   1:  PR[GP1:91,2] = PR[GP1:90,2] + 83.259;
   1:L PR[91] 10mm/sec FINE;
   1:  PR[GP1:91,1] = PR[GP1:90,1] + 112.743;
   1:  PR[GP1:91,2] = PR[GP1:90,2] + 83.554;
   1:L PR[91] 10mm/sec FINE;
   1:  PR[GP1:91,1] = PR[GP1:90,1] + 113.712;
   1:  PR[GP1:91,2] = PR[GP1:90,2] + 83.818;
   1:L PR[91] 10mm/sec FINE;
   1:  PR[GP1:91,1] = PR[GP1:90,1] + 115.940;
   1:  PR[GP1:91,2] = PR[GP1:90,2] + 84.645;
   1:L PR[91] 10mm/sec FINE;
   1:  PR[GP1:91,1] = PR[GP1:90,1] + 116.212;
   1:  PR[GP1:91,2] = PR[GP1:90,2] + 84.770;
   1:L PR[91] 10mm/sec FINE;
   1:  PR[GP1:91,1] = PR[GP1:90,1] + 117.703;
   1:  PR[GP1:91,2] = PR[GP1:90,2] + 85.648;
   1:L PR[91] 10mm/sec FINE;
   1:  PR[GP1:91,1] = PR[GP1:90,1] + 118.561;
   1:  PR[GP1:91,2] = PR[GP1:90,2] + 86.133;
   1:L PR[91] 10mm/sec FINE;
   1:  PR[GP1:91,1] = PR[GP1:90,1] + 118.735;
   1:  PR[GP1:91,2] = PR[GP1:90,2] + 86.244;
   1:L PR[91] 10mm/sec FINE;
   1:  PR[GP1:91,1] = PR[GP1:90,1] + 120.632;
   1:  PR[GP1:91,2] = PR[GP1:90,2] + 87.854;
   1:L PR[91] 10mm/sec FINE;
   1:  PR[GP1:91,1] = PR[GP1:90,1] + 121.019;
   1:  PR[GP1:91,2] = PR[GP1:90,2] + 88.214;
   1:L PR[91] 10mm/sec FINE;
   1:  PR[GP1:91,1] = PR[GP1:90,1] + 122.487;
   1:  PR[GP1:91,2] = PR[GP1:90,2] + 90.064;
   1:L PR[91] 10mm/sec FINE;
   1:  PR[GP1:91,1] = PR[GP1:90,1] + 122.811;
   1:  PR[GP1:91,2] = PR[GP1:90,2] + 90.502;
   1:L PR[91] 10mm/sec FINE;
   1:  PR[GP1:91,1] = PR[GP1:90,1] + 124.129;
   1:  PR[GP1:91,2] = PR[GP1:90,2] + 93.056;
   1:L PR[91] 10mm/sec FINE;
   1:  PR[GP1:91,1] = PR[GP1:90,1] + 124.938;
   1:  PR[GP1:91,2] = PR[GP1:90,2] + 95.541;
   1:L PR[91] 10mm/sec FINE;
   1:  PR[GP1:91,1] = PR[GP1:90,1] + 125.057;
   1:  PR[GP1:91,2] = PR[GP1:90,2] + 95.951;
   1:L PR[91] 10mm/sec FINE;
   1:  PR[GP1:91,1] = PR[GP1:90,1] + 125.342;
   1:  PR[GP1:91,2] = PR[GP1:90,2] + 97.859;
   1:L PR[91] 10mm/sec FINE;
   1:  PR[GP1:91,1] = PR[GP1:90,1] + 125.480;
   1:  PR[GP1:91,2] = PR[GP1:90,2] + 98.990;
   1:L PR[91] 10mm/sec FINE;
   1:  PR[GP1:91,1] = PR[GP1:90,1] + 125.345;
   1:  PR[GP1:91,2] = PR[GP1:90,2] + 102.010;
   1:L PR[91] 10mm/sec FINE;
   1:  PR[GP1:91,1] = PR[GP1:90,1] + 124.566;
   1:  PR[GP1:91,2] = PR[GP1:90,2] + 106.056;
   1:L PR[91] 10mm/sec FINE;
   1:  PR[GP1:91,1] = PR[GP1:90,1] + 123.318;
   1:  PR[GP1:91,2] = PR[GP1:90,2] + 109.272;
   1:L PR[91] 10mm/sec FINE;
   1:  PR[GP1:91,1] = PR[GP1:90,1] + 123.094;
   1:  PR[GP1:91,2] = PR[GP1:90,2] + 109.898;
   1:L PR[91] 10mm/sec FINE;
   1:  PR[GP1:91,1] = PR[GP1:90,1] + 121.848;
   1:  PR[GP1:91,2] = PR[GP1:90,2] + 112.039;
   1:L PR[91] 10mm/sec FINE;
   1:  PR[GP1:91,1] = PR[GP1:90,1] + 121.030;
   1:  PR[GP1:91,2] = PR[GP1:90,2] + 113.377;
   1:L PR[91] 10mm/sec FINE;
   1:  PR[GP1:91,1] = PR[GP1:90,1] + 120.172;
   1:  PR[GP1:91,2] = PR[GP1:90,2] + 114.372;
   1:L PR[91] 10mm/sec FINE;
   1:  PR[GP1:91,1] = PR[GP1:90,1] + 118.405;
   1:  PR[GP1:91,2] = PR[GP1:90,2] + 116.351;
   1:L PR[91] 10mm/sec FINE;
   1:  PR[GP1:91,1] = PR[GP1:90,1] + 115.401;
   1:  PR[GP1:91,2] = PR[GP1:90,2] + 118.708;
   1:L PR[91] 10mm/sec FINE;
   1:  PR[GP1:91,1] = PR[GP1:90,1] + 112.132;
   1:  PR[GP1:91,2] = PR[GP1:90,2] + 120.393;
   1:L PR[91] 10mm/sec FINE;
   1:  PR[GP1:91,1] = PR[GP1:90,1] + 108.661;
   1:  PR[GP1:91,2] = PR[GP1:90,2] + 121.393;
   1:L PR[91] 10mm/sec FINE;
   1:  PR[GP1:91,1] = PR[GP1:90,1] + 105.193;
   1:  PR[GP1:91,2] = PR[GP1:90,2] + 121.666;
   1:L PR[91] 10mm/sec FINE;
   1:  PR[GP1:91,1] = PR[GP1:90,1] + 101.643;
   1:  PR[GP1:91,2] = PR[GP1:90,2] + 121.281;
   1:L PR[91] 10mm/sec FINE;
   1:  PR[GP1:91,1] = PR[GP1:90,1] + 100.779;
   1:  PR[GP1:91,2] = PR[GP1:90,2] + 121.069;
   1:L PR[91] 10mm/sec FINE;
   1:  PR[GP1:91,1] = PR[GP1:90,1] + 99.835;
   1:  PR[GP1:91,2] = PR[GP1:90,2] + 121.020;
   1:L PR[91] 10mm/sec FINE;
   1:  PR[GP1:91,1] = PR[GP1:90,1] + 98.995;
   1:  PR[GP1:91,2] = PR[GP1:90,2] + 121.119;
   1:L PR[91] 10mm/sec FINE;
   1:  PR[GP1:91,1] = PR[GP1:90,1] + 98.220;
   1:  PR[GP1:91,2] = PR[GP1:90,2] + 121.182;
   1:L PR[91] 10mm/sec FINE;
   1:  PR[GP1:91,1] = PR[GP1:90,1] + 96.287;
   1:  PR[GP1:91,2] = PR[GP1:90,2] + 121.191;
   1:L PR[91] 10mm/sec FINE;
   1:  PR[GP1:91,1] = PR[GP1:90,1] + 93.391;
   1:  PR[GP1:91,2] = PR[GP1:90,2] + 121.272;
   1:L PR[91] 10mm/sec FINE;
   1:  PR[GP1:91,1] = PR[GP1:90,1] + 92.590;
   1:  PR[GP1:91,2] = PR[GP1:90,2] + 121.132;
   1:L PR[91] 10mm/sec FINE;
   1:  PR[GP1:91,1] = PR[GP1:90,1] + 88.982;
   1:  PR[GP1:91,2] = PR[GP1:90,2] + 120.605;
   1:L PR[91] 10mm/sec FINE;
   1:  PR[GP1:91,1] = PR[GP1:90,1] + 85.063;
   1:  PR[GP1:91,2] = PR[GP1:90,2] + 119.167;
   1:L PR[91] 10mm/sec FINE;
   1:  PR[GP1:91,1] = PR[GP1:90,1] + 84.544;
   1:  PR[GP1:91,2] = PR[GP1:90,2] + 118.898;
   1:L PR[91] 10mm/sec FINE;
   1:  PR[GP1:91,1] = PR[GP1:90,1] + 82.035;
   1:  PR[GP1:91,2] = PR[GP1:90,2] + 117.331;
   1:L PR[91] 10mm/sec FINE;
   1:  PR[GP1:91,1] = PR[GP1:90,1] + 81.304;
   1:  PR[GP1:91,2] = PR[GP1:90,2] + 116.806;
   1:L PR[91] 10mm/sec FINE;
   1:  PR[GP1:91,1] = PR[GP1:90,1] + 80.562;
   1:  PR[GP1:91,2] = PR[GP1:90,2] + 116.069;
   1:L PR[91] 10mm/sec FINE;
   1:  PR[GP1:91,1] = PR[GP1:90,1] + 78.972;
   1:  PR[GP1:91,2] = PR[GP1:90,2] + 114.442;
   1:L PR[91] 10mm/sec FINE;
   1:  PR[GP1:91,1] = PR[GP1:90,1] + 78.265;
   1:  PR[GP1:91,2] = PR[GP1:90,2] + 113.439;
   1:L PR[91] 10mm/sec FINE;
   1:  PR[GP1:91,1] = PR[GP1:90,1] + 77.341;
   1:  PR[GP1:91,2] = PR[GP1:90,2] + 111.823;
   1:L PR[91] 10mm/sec FINE;
   1:  PR[GP1:91,1] = PR[GP1:90,1] + 76.778;
   1:  PR[GP1:91,2] = PR[GP1:90,2] + 110.650;
   1:L PR[91] 10mm/sec FINE;
   1:  PR[GP1:91,1] = PR[GP1:90,1] + 76.425;
   1:  PR[GP1:91,2] = PR[GP1:90,2] + 109.445;
   1:L PR[91] 10mm/sec FINE;
   1:  PR[GP1:91,1] = PR[GP1:90,1] + 75.965;
   1:  PR[GP1:91,2] = PR[GP1:90,2] + 107.786;
   1:L PR[91] 10mm/sec FINE;
   1:  PR[GP1:91,1] = PR[GP1:90,1] + 75.851;
   1:  PR[GP1:91,2] = PR[GP1:90,2] + 106.711;
   1:L PR[91] 10mm/sec FINE;
   1:  PR[GP1:91,1] = PR[GP1:90,1] + 75.937;
   1:  PR[GP1:91,2] = PR[GP1:90,2] + 105.751;
   1:L PR[91] 10mm/sec FINE;
   1:  PR[GP1:91,1] = PR[GP1:90,1] + 75.997;
   1:  PR[GP1:91,2] = PR[GP1:90,2] + 103.837;
   1:L PR[91] 10mm/sec FINE;
   1:  PR[GP1:91,1] = PR[GP1:90,1] + 76.342;
   1:  PR[GP1:91,2] = PR[GP1:90,2] + 102.431;
   1:L PR[91] 10mm/sec FINE;
   1:  PR[GP1:91,1] = PR[GP1:90,1] + 76.426;
   1:  PR[GP1:91,2] = PR[GP1:90,2] + 102.023;
   1:L PR[91] 10mm/sec FINE;
   1:  PR[GP1:91,1] = PR[GP1:90,1] + 77.101;
   1:  PR[GP1:91,2] = PR[GP1:90,2] + 99.860;
   1:L PR[91] 10mm/sec FINE;
   1:  PR[GP1:91,1] = PR[GP1:90,1] + 77.622;
   1:  PR[GP1:91,2] = PR[GP1:90,2] + 98.620;
   1:L PR[91] 10mm/sec FINE;
   1:  PR[GP1:91,1] = PR[GP1:90,1] + 79.282;
   1:  PR[GP1:91,2] = PR[GP1:90,2] + 95.865;
   1:L PR[91] 10mm/sec FINE;
   1:  PR[GP1:91,1] = PR[GP1:90,1] + 79.773;
   1:  PR[GP1:91,2] = PR[GP1:90,2] + 95.104;
   1:L PR[91] 10mm/sec FINE;
   1:  PR[GP1:91,1] = PR[GP1:90,1] + 80.593;
   1:  PR[GP1:91,2] = PR[GP1:90,2] + 94.827;
   1:  PR[GP1:91,3] = PR[GP1:90,3] + 49.900;
   1:L PR[91] 10mm/sec FINE;
   1:  PR[GP1:91,1] = PR[GP1:90,1] + 80.890;
   1:  PR[GP1:91,2] = PR[GP1:90,2] + 94.492;
   1:L PR[91] 10mm/sec FINE;
   1:  PR[GP1:91,1] = PR[GP1:90,1] + 82.940;
   1:  PR[GP1:91,2] = PR[GP1:90,2] + 92.398;
   1:L PR[91] 10mm/sec FINE;
   1:  PR[GP1:91,1] = PR[GP1:90,1] + 84.017;
   1:  PR[GP1:91,2] = PR[GP1:90,2] + 91.208;
   1:L PR[91] 10mm/sec FINE;
   1:  PR[GP1:91,1] = PR[GP1:90,1] + 84.296;
   1:  PR[GP1:91,2] = PR[GP1:90,2] + 90.928;
   1:L PR[91] 10mm/sec FINE;
   1:  PR[GP1:91,1] = PR[GP1:90,1] + 87.656;
   1:  PR[GP1:91,2] = PR[GP1:90,2] + 88.402;
   1:L PR[91] 10mm/sec FINE;
   1:  PR[GP1:91,1] = PR[GP1:90,1] + 89.155;
   1:  PR[GP1:91,2] = PR[GP1:90,2] + 87.392;
   1:L PR[91] 10mm/sec FINE;
   1:  PR[GP1:91,1] = PR[GP1:90,1] + 91.747;
   1:  PR[GP1:91,2] = PR[GP1:90,2] + 86.090;
   1:L PR[91] 10mm/sec FINE;
   1:  PR[GP1:91,1] = PR[GP1:90,1] + 94.865;
   1:  PR[GP1:91,2] = PR[GP1:90,2] + 84.731;
   1:L PR[91] 10mm/sec FINE;
   1:  PR[GP1:91,1] = PR[GP1:90,1] + 96.205;
   1:  PR[GP1:91,2] = PR[GP1:90,2] + 84.332;
   1:L PR[91] 10mm/sec FINE;
   1:  PR[GP1:91,1] = PR[GP1:90,1] + 100.593;
   1:  PR[GP1:91,2] = PR[GP1:90,2] + 83.301;
   1:L PR[91] 10mm/sec FINE;
   1:  PR[GP1:91,1] = PR[GP1:90,1] + 100.999;
   1:  PR[GP1:91,2] = PR[GP1:90,2] + 83.182;
   1:L PR[91] 10mm/sec FINE;
   1:  PR[GP1:91,1] = PR[GP1:90,1] + 101.131;
   1:  PR[GP1:91,2] = PR[GP1:90,2] + 83.162;
   1:L PR[91] 10mm/sec FINE;
   1:  PR[GP1:91,1] = PR[GP1:90,1] + 106.159;
   1:  PR[GP1:91,2] = PR[GP1:90,2] + 82.678;
   1:L PR[91] 10mm/sec FINE;
   1:  PR[GP1:91,1] = PR[GP1:90,1] + 106.235;
   1:  PR[GP1:91,2] = PR[GP1:90,2] + 82.719;
   1:L PR[91] 10mm/sec FINE;
   1:  PR[GP1:91,1] = PR[GP1:90,1] + 106.414;
   1:  PR[GP1:91,2] = PR[GP1:90,2] + 82.742;
   1:L PR[91] 10mm/sec FINE;
   1:  PR[GP1:91,1] = PR[GP1:90,1] + 108.524;
   1:  PR[GP1:91,2] = PR[GP1:90,2] + 82.645;
   1:L PR[91] 10mm/sec FINE;
   1:  PR[GP1:91,1] = PR[GP1:90,1] + 110.258;
   1:  PR[GP1:91,2] = PR[GP1:90,2] + 82.682;
   1:L PR[91] 10mm/sec FINE;
   1:  PR[GP1:91,1] = PR[GP1:90,1] + 111.088;
   1:  PR[GP1:91,2] = PR[GP1:90,2] + 82.771;
   1:L PR[91] 10mm/sec FINE;
   1:  PR[GP1:91,1] = PR[GP1:90,1] + 113.708;
   1:  PR[GP1:91,2] = PR[GP1:90,2] + 83.262;
   1:L PR[91] 10mm/sec FINE;
   1:  PR[GP1:91,1] = PR[GP1:90,1] + 116.065;
   1:  PR[GP1:91,2] = PR[GP1:90,2] + 84.075;
   1:L PR[91] 10mm/sec FINE;
   1:  PR[GP1:91,1] = PR[GP1:90,1] + 116.872;
   1:  PR[GP1:91,2] = PR[GP1:90,2] + 84.409;
   1:L PR[91] 10mm/sec FINE;
   1:  PR[GP1:91,1] = PR[GP1:90,1] + 118.292;
   1:  PR[GP1:91,2] = PR[GP1:90,2] + 85.211;
   1:L PR[91] 10mm/sec FINE;
   1:  PR[GP1:91,1] = PR[GP1:90,1] + 119.566;
   1:  PR[GP1:91,2] = PR[GP1:90,2] + 86.022;
   1:L PR[91] 10mm/sec FINE;
   1:  PR[GP1:91,1] = PR[GP1:90,1] + 120.360;
   1:  PR[GP1:91,2] = PR[GP1:90,2] + 86.697;
   1:L PR[91] 10mm/sec FINE;
   1:  PR[GP1:91,1] = PR[GP1:90,1] + 121.773;
   1:  PR[GP1:91,2] = PR[GP1:90,2] + 88.008;
   1:L PR[91] 10mm/sec FINE;
   1:  PR[GP1:91,1] = PR[GP1:90,1] + 122.249;
   1:  PR[GP1:91,2] = PR[GP1:90,2] + 88.609;
   1:L PR[91] 10mm/sec FINE;
   1:  PR[GP1:91,1] = PR[GP1:90,1] + 123.495;
   1:  PR[GP1:91,2] = PR[GP1:90,2] + 90.295;
   1:L PR[91] 10mm/sec FINE;
   1:  PR[GP1:91,1] = PR[GP1:90,1] + 123.907;
   1:  PR[GP1:91,2] = PR[GP1:90,2] + 91.089;
   1:L PR[91] 10mm/sec FINE;
   1:  PR[GP1:91,1] = PR[GP1:90,1] + 124.756;
   1:  PR[GP1:91,2] = PR[GP1:90,2] + 92.826;
   1:L PR[91] 10mm/sec FINE;
   1:  PR[GP1:91,1] = PR[GP1:90,1] + 125.224;
   1:  PR[GP1:91,2] = PR[GP1:90,2] + 94.350;
   1:L PR[91] 10mm/sec FINE;
   1:  PR[GP1:91,1] = PR[GP1:90,1] + 125.576;
   1:  PR[GP1:91,2] = PR[GP1:90,2] + 95.556;
   1:L PR[91] 10mm/sec FINE;
   1:  PR[GP1:91,1] = PR[GP1:90,1] + 125.941;
   1:  PR[GP1:91,2] = PR[GP1:90,2] + 98.478;
   1:L PR[91] 10mm/sec FINE;
   1:  PR[GP1:91,1] = PR[GP1:90,1] + 125.804;
   1:  PR[GP1:91,2] = PR[GP1:90,2] + 101.583;
   1:L PR[91] 10mm/sec FINE;
   1:  PR[GP1:91,1] = PR[GP1:90,1] + 124.955;
   1:  PR[GP1:91,2] = PR[GP1:90,2] + 105.598;
   1:L PR[91] 10mm/sec FINE;
   1:  PR[GP1:91,1] = PR[GP1:90,1] + 123.477;
   1:  PR[GP1:91,2] = PR[GP1:90,2] + 109.457;
   1:L PR[91] 10mm/sec FINE;
   1:  PR[GP1:91,1] = PR[GP1:90,1] + 122.292;
   1:  PR[GP1:91,2] = PR[GP1:90,2] + 111.358;
   1:L PR[91] 10mm/sec FINE;
   1:  PR[GP1:91,1] = PR[GP1:90,1] + 121.340;
   1:  PR[GP1:91,2] = PR[GP1:90,2] + 112.968;
   1:L PR[91] 10mm/sec FINE;
   1:  PR[GP1:91,1] = PR[GP1:90,1] + 119.863;
   1:  PR[GP1:91,2] = PR[GP1:90,2] + 114.680;
   1:L PR[91] 10mm/sec FINE;
   1:  PR[GP1:91,1] = PR[GP1:90,1] + 118.711;
   1:  PR[GP1:91,2] = PR[GP1:90,2] + 115.970;
   1:L PR[91] 10mm/sec FINE;
   1:  PR[GP1:91,1] = PR[GP1:90,1] + 117.699;
   1:  PR[GP1:91,2] = PR[GP1:90,2] + 116.783;
   1:L PR[91] 10mm/sec FINE;
   1:  PR[GP1:91,1] = PR[GP1:90,1] + 115.665;
   1:  PR[GP1:91,2] = PR[GP1:90,2] + 118.364;
   1:L PR[91] 10mm/sec FINE;
   1:  PR[GP1:91,1] = PR[GP1:90,1] + 112.340;
   1:  PR[GP1:91,2] = PR[GP1:90,2] + 120.086;
   1:L PR[91] 10mm/sec FINE;
   1:  PR[GP1:91,1] = PR[GP1:90,1] + 108.882;
   1:  PR[GP1:91,2] = PR[GP1:90,2] + 121.096;
   1:L PR[91] 10mm/sec FINE;
   1:  PR[GP1:91,1] = PR[GP1:90,1] + 107.159;
   1:  PR[GP1:91,2] = PR[GP1:90,2] + 121.264;
   1:L PR[91] 10mm/sec FINE;
   1:  PR[GP1:91,1] = PR[GP1:90,1] + 105.348;
   1:  PR[GP1:91,2] = PR[GP1:90,2] + 121.403;
   1:L PR[91] 10mm/sec FINE;
   1:  PR[GP1:91,1] = PR[GP1:90,1] + 101.771;
   1:  PR[GP1:91,2] = PR[GP1:90,2] + 121.007;
   1:L PR[91] 10mm/sec FINE;
   1:  PR[GP1:91,1] = PR[GP1:90,1] + 101.109;
   1:  PR[GP1:91,2] = PR[GP1:90,2] + 120.867;
   1:L PR[91] 10mm/sec FINE;
   1:  PR[GP1:91,1] = PR[GP1:90,1] + 100.225;
   1:  PR[GP1:91,2] = PR[GP1:90,2] + 120.820;
   1:L PR[91] 10mm/sec FINE;
   1:  PR[GP1:91,1] = PR[GP1:90,1] + 99.430;
   1:  PR[GP1:91,2] = PR[GP1:90,2] + 120.900;
   1:L PR[91] 10mm/sec FINE;
   1:  PR[GP1:91,1] = PR[GP1:90,1] + 98.861;
   1:  PR[GP1:91,2] = PR[GP1:90,2] + 120.932;
   1:L PR[91] 10mm/sec FINE;
   1:  PR[GP1:91,1] = PR[GP1:90,1] + 96.648;
   1:  PR[GP1:91,2] = PR[GP1:90,2] + 120.937;
   1:L PR[91] 10mm/sec FINE;
   1:  PR[GP1:91,1] = PR[GP1:90,1] + 94.155;
   1:  PR[GP1:91,2] = PR[GP1:90,2] + 121.007;
   1:L PR[91] 10mm/sec FINE;
   1:  PR[GP1:91,1] = PR[GP1:90,1] + 92.956;
   1:  PR[GP1:91,2] = PR[GP1:90,2] + 120.798;
   1:L PR[91] 10mm/sec FINE;
   1:  PR[GP1:91,1] = PR[GP1:90,1] + 89.736;
   1:  PR[GP1:91,2] = PR[GP1:90,2] + 120.328;
   1:L PR[91] 10mm/sec FINE;
   1:  PR[GP1:91,1] = PR[GP1:90,1] + 89.390;
   1:  PR[GP1:91,2] = PR[GP1:90,2] + 120.196;
   1:L PR[91] 10mm/sec FINE;
   1:  PR[GP1:91,1] = PR[GP1:90,1] + 87.501;
   1:  PR[GP1:91,2] = PR[GP1:90,2] + 119.540;
   1:L PR[91] 10mm/sec FINE;
   1:  PR[GP1:91,1] = PR[GP1:90,1] + 85.774;
   1:  PR[GP1:91,2] = PR[GP1:90,2] + 118.905;
   1:L PR[91] 10mm/sec FINE;
   1:  PR[GP1:91,1] = PR[GP1:90,1] + 85.558;
   1:  PR[GP1:91,2] = PR[GP1:90,2] + 118.793;
   1:L PR[91] 10mm/sec FINE;
   1:  PR[GP1:91,1] = PR[GP1:90,1] + 82.642;
   1:  PR[GP1:91,2] = PR[GP1:90,2] + 116.972;
   1:L PR[91] 10mm/sec FINE;
   1:  PR[GP1:91,1] = PR[GP1:90,1] + 82.152;
   1:  PR[GP1:91,2] = PR[GP1:90,2] + 116.620;
   1:L PR[91] 10mm/sec FINE;
   1:  PR[GP1:91,1] = PR[GP1:90,1] + 79.714;
   1:  PR[GP1:91,2] = PR[GP1:90,2] + 114.140;
   1:L PR[91] 10mm/sec FINE;
   1:  PR[GP1:91,1] = PR[GP1:90,1] + 79.187;
   1:  PR[GP1:91,2] = PR[GP1:90,2] + 113.393;
   1:L PR[91] 10mm/sec FINE;
   1:  PR[GP1:91,1] = PR[GP1:90,1] + 78.039;
   1:  PR[GP1:91,2] = PR[GP1:90,2] + 111.385;
   1:L PR[91] 10mm/sec FINE;
   1:  PR[GP1:91,1] = PR[GP1:90,1] + 77.606;
   1:  PR[GP1:91,2] = PR[GP1:90,2] + 110.484;
   1:L PR[91] 10mm/sec FINE;
   1:  PR[GP1:91,1] = PR[GP1:90,1] + 76.754;
   1:  PR[GP1:91,2] = PR[GP1:90,2] + 107.459;
   1:L PR[91] 10mm/sec FINE;
   1:  PR[GP1:91,1] = PR[GP1:90,1] + 76.666;
   1:  PR[GP1:91,2] = PR[GP1:90,2] + 106.641;
   1:L PR[91] 10mm/sec FINE;
   1:  PR[GP1:91,1] = PR[GP1:90,1] + 76.733;
   1:  PR[GP1:91,2] = PR[GP1:90,2] + 105.905;
   1:L PR[91] 10mm/sec FINE;
   1:  PR[GP1:91,1] = PR[GP1:90,1] + 76.806;
   1:  PR[GP1:91,2] = PR[GP1:90,2] + 103.545;
   1:L PR[91] 10mm/sec FINE;
   1:  PR[GP1:91,1] = PR[GP1:90,1] + 77.058;
   1:  PR[GP1:91,2] = PR[GP1:90,2] + 102.521;
   1:L PR[91] 10mm/sec FINE;
   1:  PR[GP1:91,1] = PR[GP1:90,1] + 77.159;
   1:  PR[GP1:91,2] = PR[GP1:90,2] + 102.032;
   1:L PR[91] 10mm/sec FINE;
   1:  PR[GP1:91,1] = PR[GP1:90,1] + 77.965;
   1:  PR[GP1:91,2] = PR[GP1:90,2] + 99.443;
   1:L PR[91] 10mm/sec FINE;
   1:  PR[GP1:91,1] = PR[GP1:90,1] + 78.366;
   1:  PR[GP1:91,2] = PR[GP1:90,2] + 98.491;
   1:L PR[91] 10mm/sec FINE;
   1:  PR[GP1:91,1] = PR[GP1:90,1] + 80.302;
   1:  PR[GP1:91,2] = PR[GP1:90,2] + 95.279;
   1:L PR[91] 10mm/sec FINE;
   1:  PR[GP1:91,1] = PR[GP1:90,1] + 81.413;
   1:  PR[GP1:91,2] = PR[GP1:90,2] + 94.550;
   1:  PR[GP1:91,3] = PR[GP1:90,3] + 50.900;
   1:L PR[91] 10mm/sec FINE;
   1:  PR[GP1:91,1] = PR[GP1:90,1] + 81.505;
   1:  PR[GP1:91,2] = PR[GP1:90,2] + 94.447;
   1:L PR[91] 10mm/sec FINE;
   1:  PR[GP1:91,1] = PR[GP1:90,1] + 82.201;
   1:  PR[GP1:91,2] = PR[GP1:90,2] + 93.736;
   1:L PR[91] 10mm/sec FINE;
   1:  PR[GP1:91,1] = PR[GP1:90,1] + 84.569;
   1:  PR[GP1:91,2] = PR[GP1:90,2] + 91.119;
   1:L PR[91] 10mm/sec FINE;
   1:  PR[GP1:91,1] = PR[GP1:90,1] + 85.199;
   1:  PR[GP1:91,2] = PR[GP1:90,2] + 90.489;
   1:L PR[91] 10mm/sec FINE;
   1:  PR[GP1:91,1] = PR[GP1:90,1] + 88.167;
   1:  PR[GP1:91,2] = PR[GP1:90,2] + 88.258;
   1:L PR[91] 10mm/sec FINE;
   1:  PR[GP1:91,1] = PR[GP1:90,1] + 90.100;
   1:  PR[GP1:91,2] = PR[GP1:90,2] + 86.955;
   1:L PR[91] 10mm/sec FINE;
   1:  PR[GP1:91,1] = PR[GP1:90,1] + 92.234;
   1:  PR[GP1:91,2] = PR[GP1:90,2] + 85.883;
   1:L PR[91] 10mm/sec FINE;
   1:  PR[GP1:91,1] = PR[GP1:90,1] + 95.849;
   1:  PR[GP1:91,2] = PR[GP1:90,2] + 84.307;
   1:L PR[91] 10mm/sec FINE;
   1:  PR[GP1:91,1] = PR[GP1:90,1] + 96.686;
   1:  PR[GP1:91,2] = PR[GP1:90,2] + 84.058;
   1:L PR[91] 10mm/sec FINE;
   1:  PR[GP1:91,1] = PR[GP1:90,1] + 99.448;
   1:  PR[GP1:91,2] = PR[GP1:90,2] + 83.409;
   1:L PR[91] 10mm/sec FINE;
   1:  PR[GP1:91,1] = PR[GP1:90,1] + 101.663;
   1:  PR[GP1:91,2] = PR[GP1:90,2] + 82.761;
   1:L PR[91] 10mm/sec FINE;
   1:  PR[GP1:91,1] = PR[GP1:90,1] + 102.452;
   1:  PR[GP1:91,2] = PR[GP1:90,2] + 82.642;
   1:L PR[91] 10mm/sec FINE;
   1:  PR[GP1:91,1] = PR[GP1:90,1] + 106.815;
   1:  PR[GP1:91,2] = PR[GP1:90,2] + 82.221;
   1:L PR[91] 10mm/sec FINE;
   1:  PR[GP1:91,1] = PR[GP1:90,1] + 106.881;
   1:  PR[GP1:91,2] = PR[GP1:90,2] + 82.256;
   1:L PR[91] 10mm/sec FINE;
   1:  PR[GP1:91,1] = PR[GP1:90,1] + 107.240;
   1:  PR[GP1:91,2] = PR[GP1:90,2] + 82.296;
   1:L PR[91] 10mm/sec FINE;
   1:  PR[GP1:91,1] = PR[GP1:90,1] + 108.414;
   1:  PR[GP1:91,2] = PR[GP1:90,2] + 82.240;
   1:L PR[91] 10mm/sec FINE;
   1:  PR[GP1:91,1] = PR[GP1:90,1] + 111.163;
   1:  PR[GP1:91,2] = PR[GP1:90,2] + 82.299;
   1:L PR[91] 10mm/sec FINE;
   1:  PR[GP1:91,1] = PR[GP1:90,1] + 113.486;
   1:  PR[GP1:91,2] = PR[GP1:90,2] + 82.673;
   1:L PR[91] 10mm/sec FINE;
   1:  PR[GP1:91,1] = PR[GP1:90,1] + 114.692;
   1:  PR[GP1:91,2] = PR[GP1:90,2] + 82.952;
   1:L PR[91] 10mm/sec FINE;
   1:  PR[GP1:91,1] = PR[GP1:90,1] + 115.821;
   1:  PR[GP1:91,2] = PR[GP1:90,2] + 83.341;
   1:L PR[91] 10mm/sec FINE;
   1:  PR[GP1:91,1] = PR[GP1:90,1] + 117.782;
   1:  PR[GP1:91,2] = PR[GP1:90,2] + 84.153;
   1:L PR[91] 10mm/sec FINE;
   1:  PR[GP1:91,1] = PR[GP1:90,1] + 118.023;
   1:  PR[GP1:91,2] = PR[GP1:90,2] + 84.289;
   1:L PR[91] 10mm/sec FINE;
   1:  PR[GP1:91,1] = PR[GP1:90,1] + 118.960;
   1:  PR[GP1:91,2] = PR[GP1:90,2] + 84.886;
   1:L PR[91] 10mm/sec FINE;
   1:  PR[GP1:91,1] = PR[GP1:90,1] + 120.290;
   1:  PR[GP1:91,2] = PR[GP1:90,2] + 85.703;
   1:L PR[91] 10mm/sec FINE;
   1:  PR[GP1:91,1] = PR[GP1:90,1] + 122.398;
   1:  PR[GP1:91,2] = PR[GP1:90,2] + 87.611;
   1:L PR[91] 10mm/sec FINE;
   1:  PR[GP1:91,1] = PR[GP1:90,1] + 122.951;
   1:  PR[GP1:91,2] = PR[GP1:90,2] + 88.334;
   1:L PR[91] 10mm/sec FINE;
   1:  PR[GP1:91,1] = PR[GP1:90,1] + 124.115;
   1:  PR[GP1:91,2] = PR[GP1:90,2] + 89.911;
   1:L PR[91] 10mm/sec FINE;
   1:  PR[GP1:91,1] = PR[GP1:90,1] + 125.376;
   1:  PR[GP1:91,2] = PR[GP1:90,2] + 92.527;
   1:L PR[91] 10mm/sec FINE;
   1:  PR[GP1:91,1] = PR[GP1:90,1] + 126.161;
   1:  PR[GP1:91,2] = PR[GP1:90,2] + 95.296;
   1:L PR[91] 10mm/sec FINE;
   1:  PR[GP1:91,1] = PR[GP1:90,1] + 126.489;
   1:  PR[GP1:91,2] = PR[GP1:90,2] + 98.156;
   1:L PR[91] 10mm/sec FINE;
   1:  PR[GP1:91,1] = PR[GP1:90,1] + 126.285;
   1:  PR[GP1:91,2] = PR[GP1:90,2] + 101.175;
   1:L PR[91] 10mm/sec FINE;
   1:  PR[GP1:91,1] = PR[GP1:90,1] + 126.019;
   1:  PR[GP1:91,2] = PR[GP1:90,2] + 102.333;
   1:L PR[91] 10mm/sec FINE;
   1:  PR[GP1:91,1] = PR[GP1:90,1] + 125.412;
   1:  PR[GP1:91,2] = PR[GP1:90,2] + 105.182;
   1:L PR[91] 10mm/sec FINE;
   1:  PR[GP1:91,1] = PR[GP1:90,1] + 124.598;
   1:  PR[GP1:91,2] = PR[GP1:90,2] + 107.148;
   1:L PR[91] 10mm/sec FINE;
   1:  PR[GP1:91,1] = PR[GP1:90,1] + 123.882;
   1:  PR[GP1:91,2] = PR[GP1:90,2] + 109.022;
   1:L PR[91] 10mm/sec FINE;
   1:  PR[GP1:91,1] = PR[GP1:90,1] + 122.963;
   1:  PR[GP1:91,2] = PR[GP1:90,2] + 110.530;
   1:L PR[91] 10mm/sec FINE;
   1:  PR[GP1:91,1] = PR[GP1:90,1] + 121.690;
   1:  PR[GP1:91,2] = PR[GP1:90,2] + 112.553;
   1:L PR[91] 10mm/sec FINE;
   1:  PR[GP1:91,1] = PR[GP1:90,1] + 120.900;
   1:  PR[GP1:91,2] = PR[GP1:90,2] + 113.428;
   1:L PR[91] 10mm/sec FINE;
   1:  PR[GP1:91,1] = PR[GP1:90,1] + 119.555;
   1:  PR[GP1:91,2] = PR[GP1:90,2] + 114.988;
   1:L PR[91] 10mm/sec FINE;
   1:  PR[GP1:91,1] = PR[GP1:90,1] + 119.017;
   1:  PR[GP1:91,2] = PR[GP1:90,2] + 115.589;
   1:L PR[91] 10mm/sec FINE;
   1:  PR[GP1:91,1] = PR[GP1:90,1] + 117.307;
   1:  PR[GP1:91,2] = PR[GP1:90,2] + 116.963;
   1:L PR[91] 10mm/sec FINE;
   1:  PR[GP1:91,1] = PR[GP1:90,1] + 115.959;
   1:  PR[GP1:91,2] = PR[GP1:90,2] + 118.011;
   1:L PR[91] 10mm/sec FINE;
   1:  PR[GP1:91,1] = PR[GP1:90,1] + 114.604;
   1:  PR[GP1:91,2] = PR[GP1:90,2] + 118.733;
   1:L PR[91] 10mm/sec FINE;
   1:  PR[GP1:91,1] = PR[GP1:90,1] + 112.611;
   1:  PR[GP1:91,2] = PR[GP1:90,2] + 119.759;
   1:L PR[91] 10mm/sec FINE;
   1:  PR[GP1:91,1] = PR[GP1:90,1] + 111.126;
   1:  PR[GP1:91,2] = PR[GP1:90,2] + 120.214;
   1:L PR[91] 10mm/sec FINE;
   1:  PR[GP1:91,1] = PR[GP1:90,1] + 109.106;
   1:  PR[GP1:91,2] = PR[GP1:90,2] + 120.799;
   1:L PR[91] 10mm/sec FINE;
   1:  PR[GP1:91,1] = PR[GP1:90,1] + 105.501;
   1:  PR[GP1:91,2] = PR[GP1:90,2] + 121.139;
   1:L PR[91] 10mm/sec FINE;
   1:  PR[GP1:91,1] = PR[GP1:90,1] + 101.901;
   1:  PR[GP1:91,2] = PR[GP1:90,2] + 120.734;
   1:L PR[91] 10mm/sec FINE;
   1:  PR[GP1:91,1] = PR[GP1:90,1] + 101.457;
   1:  PR[GP1:91,2] = PR[GP1:90,2] + 120.651;
   1:L PR[91] 10mm/sec FINE;
   1:  PR[GP1:91,1] = PR[GP1:90,1] + 100.629;
   1:  PR[GP1:91,2] = PR[GP1:90,2] + 120.610;
   1:L PR[91] 10mm/sec FINE;
   1:  PR[GP1:91,1] = PR[GP1:90,1] + 99.634;
   1:  PR[GP1:91,2] = PR[GP1:90,2] + 120.677;
   1:L PR[91] 10mm/sec FINE;
   1:  PR[GP1:91,1] = PR[GP1:90,1] + 97.009;
   1:  PR[GP1:91,2] = PR[GP1:90,2] + 120.683;
   1:L PR[91] 10mm/sec FINE;
   1:  PR[GP1:91,1] = PR[GP1:90,1] + 94.919;
   1:  PR[GP1:91,2] = PR[GP1:90,2] + 120.742;
   1:L PR[91] 10mm/sec FINE;
   1:  PR[GP1:91,1] = PR[GP1:90,1] + 93.322;
   1:  PR[GP1:91,2] = PR[GP1:90,2] + 120.463;
   1:L PR[91] 10mm/sec FINE;
   1:  PR[GP1:91,1] = PR[GP1:90,1] + 90.494;
   1:  PR[GP1:91,2] = PR[GP1:90,2] + 120.050;
   1:L PR[91] 10mm/sec FINE;
   1:  PR[GP1:91,1] = PR[GP1:90,1] + 89.777;
   1:  PR[GP1:91,2] = PR[GP1:90,2] + 119.776;
   1:L PR[91] 10mm/sec FINE;
   1:  PR[GP1:91,1] = PR[GP1:90,1] + 86.501;
   1:  PR[GP1:91,2] = PR[GP1:90,2] + 118.638;
   1:L PR[91] 10mm/sec FINE;
   1:  PR[GP1:91,1] = PR[GP1:90,1] + 83.250;
   1:  PR[GP1:91,2] = PR[GP1:90,2] + 116.612;
   1:L PR[91] 10mm/sec FINE;
   1:  PR[GP1:91,1] = PR[GP1:90,1] + 82.999;
   1:  PR[GP1:91,2] = PR[GP1:90,2] + 116.432;
   1:L PR[91] 10mm/sec FINE;
   1:  PR[GP1:91,1] = PR[GP1:90,1] + 80.457;
   1:  PR[GP1:91,2] = PR[GP1:90,2] + 113.839;
   1:L PR[91] 10mm/sec FINE;
   1:  PR[GP1:91,1] = PR[GP1:90,1] + 80.109;
   1:  PR[GP1:91,2] = PR[GP1:90,2] + 113.346;
   1:L PR[91] 10mm/sec FINE;
   1:  PR[GP1:91,1] = PR[GP1:90,1] + 78.738;
   1:  PR[GP1:91,2] = PR[GP1:90,2] + 110.947;
   1:L PR[91] 10mm/sec FINE;
   1:  PR[GP1:91,1] = PR[GP1:90,1] + 78.434;
   1:  PR[GP1:91,2] = PR[GP1:90,2] + 110.316;
   1:L PR[91] 10mm/sec FINE;
   1:  PR[GP1:91,1] = PR[GP1:90,1] + 77.542;
   1:  PR[GP1:91,2] = PR[GP1:90,2] + 107.134;
   1:L PR[91] 10mm/sec FINE;
   1:  PR[GP1:91,1] = PR[GP1:90,1] + 77.482;
   1:  PR[GP1:91,2] = PR[GP1:90,2] + 106.571;
   1:L PR[91] 10mm/sec FINE;
   1:  PR[GP1:91,1] = PR[GP1:90,1] + 77.528;
   1:  PR[GP1:91,2] = PR[GP1:90,2] + 106.060;
   1:L PR[91] 10mm/sec FINE;
   1:  PR[GP1:91,1] = PR[GP1:90,1] + 77.616;
   1:  PR[GP1:91,2] = PR[GP1:90,2] + 103.252;
   1:L PR[91] 10mm/sec FINE;
   1:  PR[GP1:91,1] = PR[GP1:90,1] + 77.773;
   1:  PR[GP1:91,2] = PR[GP1:90,2] + 102.611;
   1:L PR[91] 10mm/sec FINE;
   1:  PR[GP1:91,1] = PR[GP1:90,1] + 77.891;
   1:  PR[GP1:91,2] = PR[GP1:90,2] + 102.041;
   1:L PR[91] 10mm/sec FINE;
   1:  PR[GP1:91,1] = PR[GP1:90,1] + 78.830;
   1:  PR[GP1:91,2] = PR[GP1:90,2] + 99.027;
   1:L PR[91] 10mm/sec FINE;
   1:  PR[GP1:91,1] = PR[GP1:90,1] + 79.109;
   1:  PR[GP1:91,2] = PR[GP1:90,2] + 98.363;
   1:L PR[91] 10mm/sec FINE;
   1:  PR[GP1:91,1] = PR[GP1:90,1] + 81.321;
   1:  PR[GP1:91,2] = PR[GP1:90,2] + 94.694;
   1:L PR[91] 10mm/sec FINE;
   1:  PR[GP1:91,1] = PR[GP1:90,1] + 82.145;
   1:  PR[GP1:91,2] = PR[GP1:90,2] + 94.369;
   1:  PR[GP1:91,3] = PR[GP1:90,3] + 51.900;
   1:L PR[91] 10mm/sec FINE;
   1:  PR[GP1:91,1] = PR[GP1:90,1] + 82.254;
   1:  PR[GP1:91,2] = PR[GP1:90,2] + 94.199;
   1:L PR[91] 10mm/sec FINE;
   1:  PR[GP1:91,1] = PR[GP1:90,1] + 85.120;
   1:  PR[GP1:91,2] = PR[GP1:90,2] + 91.031;
   1:L PR[91] 10mm/sec FINE;
   1:  PR[GP1:91,1] = PR[GP1:90,1] + 86.102;
   1:  PR[GP1:91,2] = PR[GP1:90,2] + 90.051;
   1:L PR[91] 10mm/sec FINE;
   1:  PR[GP1:91,1] = PR[GP1:90,1] + 88.678;
   1:  PR[GP1:91,2] = PR[GP1:90,2] + 88.114;
   1:L PR[91] 10mm/sec FINE;
   1:  PR[GP1:91,1] = PR[GP1:90,1] + 91.045;
   1:  PR[GP1:91,2] = PR[GP1:90,2] + 86.519;
   1:L PR[91] 10mm/sec FINE;
   1:  PR[GP1:91,1] = PR[GP1:90,1] + 92.722;
   1:  PR[GP1:91,2] = PR[GP1:90,2] + 85.677;
   1:L PR[91] 10mm/sec FINE;
   1:  PR[GP1:91,1] = PR[GP1:90,1] + 96.834;
   1:  PR[GP1:91,2] = PR[GP1:90,2] + 83.883;
   1:L PR[91] 10mm/sec FINE;
   1:  PR[GP1:91,1] = PR[GP1:90,1] + 97.168;
   1:  PR[GP1:91,2] = PR[GP1:90,2] + 83.784;
   1:L PR[91] 10mm/sec FINE;
   1:  PR[GP1:91,1] = PR[GP1:90,1] + 98.302;
   1:  PR[GP1:91,2] = PR[GP1:90,2] + 83.518;
   1:L PR[91] 10mm/sec FINE;
   1:  PR[GP1:91,1] = PR[GP1:90,1] + 102.326;
   1:  PR[GP1:91,2] = PR[GP1:90,2] + 82.340;
   1:L PR[91] 10mm/sec FINE;
   1:  PR[GP1:91,1] = PR[GP1:90,1] + 103.773;
   1:  PR[GP1:91,2] = PR[GP1:90,2] + 82.121;
   1:L PR[91] 10mm/sec FINE;
   1:  PR[GP1:91,1] = PR[GP1:90,1] + 107.472;
   1:  PR[GP1:91,2] = PR[GP1:90,2] + 81.764;
   1:L PR[91] 10mm/sec FINE;
   1:  PR[GP1:91,1] = PR[GP1:90,1] + 107.523;
   1:  PR[GP1:91,2] = PR[GP1:90,2] + 81.792;
   1:L PR[91] 10mm/sec FINE;
   1:  PR[GP1:91,1] = PR[GP1:90,1] + 107.771;
   1:  PR[GP1:91,2] = PR[GP1:90,2] + 81.824;
   1:L PR[91] 10mm/sec FINE;
   1:  PR[GP1:91,1] = PR[GP1:90,1] + 108.158;
   1:  PR[GP1:91,2] = PR[GP1:90,2] + 81.838;
   1:L PR[91] 10mm/sec FINE;
   1:  PR[GP1:91,1] = PR[GP1:90,1] + 110.855;
   1:  PR[GP1:91,2] = PR[GP1:90,2] + 81.825;
   1:L PR[91] 10mm/sec FINE;
   1:  PR[GP1:91,1] = PR[GP1:90,1] + 112.218;
   1:  PR[GP1:91,2] = PR[GP1:90,2] + 81.917;
   1:L PR[91] 10mm/sec FINE;
   1:  PR[GP1:91,1] = PR[GP1:90,1] + 113.283;
   1:  PR[GP1:91,2] = PR[GP1:90,2] + 82.089;
   1:L PR[91] 10mm/sec FINE;
   1:  PR[GP1:91,1] = PR[GP1:90,1] + 115.630;
   1:  PR[GP1:91,2] = PR[GP1:90,2] + 82.625;
   1:L PR[91] 10mm/sec FINE;
   1:  PR[GP1:91,1] = PR[GP1:90,1] + 118.278;
   1:  PR[GP1:91,2] = PR[GP1:90,2] + 83.651;
   1:L PR[91] 10mm/sec FINE;
   1:  PR[GP1:91,1] = PR[GP1:90,1] + 119.737;
   1:  PR[GP1:91,2] = PR[GP1:90,2] + 84.507;
   1:L PR[91] 10mm/sec FINE;
   1:  PR[GP1:91,1] = PR[GP1:90,1] + 120.731;
   1:  PR[GP1:91,2] = PR[GP1:90,2] + 85.117;
   1:L PR[91] 10mm/sec FINE;
   1:  PR[GP1:91,1] = PR[GP1:90,1] + 122.899;
   1:  PR[GP1:91,2] = PR[GP1:90,2] + 87.029;
   1:L PR[91] 10mm/sec FINE;
   1:  PR[GP1:91,1] = PR[GP1:90,1] + 124.674;
   1:  PR[GP1:91,2] = PR[GP1:90,2] + 89.356;
   1:L PR[91] 10mm/sec FINE;
   1:  PR[GP1:91,1] = PR[GP1:90,1] + 125.978;
   1:  PR[GP1:91,2] = PR[GP1:90,2] + 92.019;
   1:L PR[91] 10mm/sec FINE;
   1:  PR[GP1:91,1] = PR[GP1:90,1] + 126.778;
   1:  PR[GP1:91,2] = PR[GP1:90,2] + 94.893;
   1:L PR[91] 10mm/sec FINE;
   1:  PR[GP1:91,1] = PR[GP1:90,1] + 127.053;
   1:  PR[GP1:91,2] = PR[GP1:90,2] + 97.848;
   1:L PR[91] 10mm/sec FINE;
   1:  PR[GP1:91,1] = PR[GP1:90,1] + 126.816;
   1:  PR[GP1:91,2] = PR[GP1:90,2] + 100.815;
   1:L PR[91] 10mm/sec FINE;
   1:  PR[GP1:91,1] = PR[GP1:90,1] + 126.066;
   1:  PR[GP1:91,2] = PR[GP1:90,2] + 103.926;
   1:L PR[91] 10mm/sec FINE;
   1:  PR[GP1:91,1] = PR[GP1:90,1] + 125.880;
   1:  PR[GP1:91,2] = PR[GP1:90,2] + 104.775;
   1:L PR[91] 10mm/sec FINE;
   1:  PR[GP1:91,1] = PR[GP1:90,1] + 124.304;
   1:  PR[GP1:91,2] = PR[GP1:90,2] + 108.591;
   1:L PR[91] 10mm/sec FINE;
   1:  PR[GP1:91,1] = PR[GP1:90,1] + 124.027;
   1:  PR[GP1:91,2] = PR[GP1:90,2] + 109.015;
   1:L PR[91] 10mm/sec FINE;
   1:  PR[GP1:91,1] = PR[GP1:90,1] + 122.838;
   1:  PR[GP1:91,2] = PR[GP1:90,2] + 110.966;
   1:L PR[91] 10mm/sec FINE;
   1:  PR[GP1:91,1] = PR[GP1:90,1] + 122.099;
   1:  PR[GP1:91,2] = PR[GP1:90,2] + 112.140;
   1:L PR[91] 10mm/sec FINE;
   1:  PR[GP1:91,1] = PR[GP1:90,1] + 119.335;
   1:  PR[GP1:91,2] = PR[GP1:90,2] + 115.207;
   1:L PR[91] 10mm/sec FINE;
   1:  PR[GP1:91,1] = PR[GP1:90,1] + 116.253;
   1:  PR[GP1:91,2] = PR[GP1:90,2] + 117.658;
   1:L PR[91] 10mm/sec FINE;
   1:  PR[GP1:91,1] = PR[GP1:90,1] + 114.109;
   1:  PR[GP1:91,2] = PR[GP1:90,2] + 118.801;
   1:L PR[91] 10mm/sec FINE;
   1:  PR[GP1:91,1] = PR[GP1:90,1] + 112.883;
   1:  PR[GP1:91,2] = PR[GP1:90,2] + 119.432;
   1:L PR[91] 10mm/sec FINE;
   1:  PR[GP1:91,1] = PR[GP1:90,1] + 110.370;
   1:  PR[GP1:91,2] = PR[GP1:90,2] + 120.201;
   1:L PR[91] 10mm/sec FINE;
   1:  PR[GP1:91,1] = PR[GP1:90,1] + 109.329;
   1:  PR[GP1:91,2] = PR[GP1:90,2] + 120.503;
   1:L PR[91] 10mm/sec FINE;
   1:  PR[GP1:91,1] = PR[GP1:90,1] + 105.720;
   1:  PR[GP1:91,2] = PR[GP1:90,2] + 120.856;
   1:L PR[91] 10mm/sec FINE;
   1:  PR[GP1:91,1] = PR[GP1:90,1] + 104.933;
   1:  PR[GP1:91,2] = PR[GP1:90,2] + 120.789;
   1:L PR[91] 10mm/sec FINE;
   1:  PR[GP1:91,1] = PR[GP1:90,1] + 102.032;
   1:  PR[GP1:91,2] = PR[GP1:90,2] + 120.461;
   1:L PR[91] 10mm/sec FINE;
   1:  PR[GP1:91,1] = PR[GP1:90,1] + 101.822;
   1:  PR[GP1:91,2] = PR[GP1:90,2] + 120.425;
   1:L PR[91] 10mm/sec FINE;
   1:  PR[GP1:91,1] = PR[GP1:90,1] + 101.047;
   1:  PR[GP1:91,2] = PR[GP1:90,2] + 120.388;
   1:L PR[91] 10mm/sec FINE;
   1:  PR[GP1:91,1] = PR[GP1:90,1] + 100.409;
   1:  PR[GP1:91,2] = PR[GP1:90,2] + 120.423;
   1:L PR[91] 10mm/sec FINE;
   1:  PR[GP1:91,1] = PR[GP1:90,1] + 97.370;
   1:  PR[GP1:91,2] = PR[GP1:90,2] + 120.429;
   1:L PR[91] 10mm/sec FINE;
   1:  PR[GP1:91,1] = PR[GP1:90,1] + 95.683;
   1:  PR[GP1:91,2] = PR[GP1:90,2] + 120.477;
   1:L PR[91] 10mm/sec FINE;
   1:  PR[GP1:91,1] = PR[GP1:90,1] + 93.687;
   1:  PR[GP1:91,2] = PR[GP1:90,2] + 120.128;
   1:L PR[91] 10mm/sec FINE;
   1:  PR[GP1:91,1] = PR[GP1:90,1] + 91.251;
   1:  PR[GP1:91,2] = PR[GP1:90,2] + 119.773;
   1:L PR[91] 10mm/sec FINE;
   1:  PR[GP1:91,1] = PR[GP1:90,1] + 90.163;
   1:  PR[GP1:91,2] = PR[GP1:90,2] + 119.356;
   1:L PR[91] 10mm/sec FINE;
   1:  PR[GP1:91,1] = PR[GP1:90,1] + 87.258;
   1:  PR[GP1:91,2] = PR[GP1:90,2] + 118.347;
   1:L PR[91] 10mm/sec FINE;
   1:  PR[GP1:91,1] = PR[GP1:90,1] + 86.872;
   1:  PR[GP1:91,2] = PR[GP1:90,2] + 118.093;
   1:L PR[91] 10mm/sec FINE;
   1:  PR[GP1:91,1] = PR[GP1:90,1] + 83.841;
   1:  PR[GP1:91,2] = PR[GP1:90,2] + 116.240;
   1:L PR[91] 10mm/sec FINE;
   1:  PR[GP1:91,1] = PR[GP1:90,1] + 81.199;
   1:  PR[GP1:91,2] = PR[GP1:90,2] + 113.538;
   1:L PR[91] 10mm/sec FINE;
   1:  PR[GP1:91,1] = PR[GP1:90,1] + 81.031;
   1:  PR[GP1:91,2] = PR[GP1:90,2] + 113.300;
   1:L PR[91] 10mm/sec FINE;
   1:  PR[GP1:91,1] = PR[GP1:90,1] + 79.436;
   1:  PR[GP1:91,2] = PR[GP1:90,2] + 110.509;
   1:L PR[91] 10mm/sec FINE;
   1:  PR[GP1:91,1] = PR[GP1:90,1] + 79.263;
   1:  PR[GP1:91,2] = PR[GP1:90,2] + 110.149;
   1:L PR[91] 10mm/sec FINE;
   1:  PR[GP1:91,1] = PR[GP1:90,1] + 78.331;
   1:  PR[GP1:91,2] = PR[GP1:90,2] + 106.808;
   1:L PR[91] 10mm/sec FINE;
   1:  PR[GP1:91,1] = PR[GP1:90,1] + 78.298;
   1:  PR[GP1:91,2] = PR[GP1:90,2] + 106.501;
   1:L PR[91] 10mm/sec FINE;
   1:  PR[GP1:91,1] = PR[GP1:90,1] + 78.324;
   1:  PR[GP1:91,2] = PR[GP1:90,2] + 106.214;
   1:L PR[91] 10mm/sec FINE;
   1:  PR[GP1:91,1] = PR[GP1:90,1] + 78.425;
   1:  PR[GP1:91,2] = PR[GP1:90,2] + 102.958;
   1:L PR[91] 10mm/sec FINE;
   1:  PR[GP1:91,1] = PR[GP1:90,1] + 78.622;
   1:  PR[GP1:91,2] = PR[GP1:90,2] + 102.052;
   1:L PR[91] 10mm/sec FINE;
   1:  PR[GP1:91,1] = PR[GP1:90,1] + 79.695;
   1:  PR[GP1:91,2] = PR[GP1:90,2] + 98.610;
   1:L PR[91] 10mm/sec FINE;
   1:  PR[GP1:91,1] = PR[GP1:90,1] + 79.853;
   1:  PR[GP1:91,2] = PR[GP1:90,2] + 98.235;
   1:L PR[91] 10mm/sec FINE;
   1:  PR[GP1:91,1] = PR[GP1:90,1] + 81.594;
   1:  PR[GP1:91,2] = PR[GP1:90,2] + 95.347;
   1:L PR[91] 10mm/sec FINE;
   1:  PR[GP1:91,1] = PR[GP1:90,1] + 83.117;
   1:  PR[GP1:91,2] = PR[GP1:90,2] + 93.767;
   1:  PR[GP1:91,3] = PR[GP1:90,3] + 52.900;
   1:L PR[91] 10mm/sec FINE;
   1:  PR[GP1:91,1] = PR[GP1:90,1] + 85.672;
   1:  PR[GP1:91,2] = PR[GP1:90,2] + 90.943;
   1:L PR[91] 10mm/sec FINE;
   1:  PR[GP1:91,1] = PR[GP1:90,1] + 87.005;
   1:  PR[GP1:91,2] = PR[GP1:90,2] + 89.612;
   1:L PR[91] 10mm/sec FINE;
   1:  PR[GP1:91,1] = PR[GP1:90,1] + 89.189;
   1:  PR[GP1:91,2] = PR[GP1:90,2] + 87.970;
   1:L PR[91] 10mm/sec FINE;
   1:  PR[GP1:91,1] = PR[GP1:90,1] + 91.990;
   1:  PR[GP1:91,2] = PR[GP1:90,2] + 86.082;
   1:L PR[91] 10mm/sec FINE;
   1:  PR[GP1:91,1] = PR[GP1:90,1] + 93.209;
   1:  PR[GP1:91,2] = PR[GP1:90,2] + 85.470;
   1:L PR[91] 10mm/sec FINE;
   1:  PR[GP1:91,1] = PR[GP1:90,1] + 97.233;
   1:  PR[GP1:91,2] = PR[GP1:90,2] + 83.715;
   1:L PR[91] 10mm/sec FINE;
   1:  PR[GP1:91,1] = PR[GP1:90,1] + 97.735;
   1:  PR[GP1:91,2] = PR[GP1:90,2] + 83.465;
   1:L PR[91] 10mm/sec FINE;
   1:  PR[GP1:91,1] = PR[GP1:90,1] + 97.922;
   1:  PR[GP1:91,2] = PR[GP1:90,2] + 83.402;
   1:L PR[91] 10mm/sec FINE;
   1:  PR[GP1:91,1] = PR[GP1:90,1] + 102.990;
   1:  PR[GP1:91,2] = PR[GP1:90,2] + 81.919;
   1:L PR[91] 10mm/sec FINE;
   1:  PR[GP1:91,1] = PR[GP1:90,1] + 105.094;
   1:  PR[GP1:91,2] = PR[GP1:90,2] + 81.600;
   1:L PR[91] 10mm/sec FINE;
   1:  PR[GP1:91,1] = PR[GP1:90,1] + 108.128;
   1:  PR[GP1:91,2] = PR[GP1:90,2] + 81.308;
   1:L PR[91] 10mm/sec FINE;
   1:  PR[GP1:91,1] = PR[GP1:90,1] + 108.166;
   1:  PR[GP1:91,2] = PR[GP1:90,2] + 81.328;
   1:L PR[91] 10mm/sec FINE;
   1:  PR[GP1:91,1] = PR[GP1:90,1] + 108.379;
   1:  PR[GP1:91,2] = PR[GP1:90,2] + 81.356;
   1:L PR[91] 10mm/sec FINE;
   1:  PR[GP1:91,1] = PR[GP1:90,1] + 108.818;
   1:  PR[GP1:91,2] = PR[GP1:90,2] + 81.372;
   1:L PR[91] 10mm/sec FINE;
   1:  PR[GP1:91,1] = PR[GP1:90,1] + 110.693;
   1:  PR[GP1:91,2] = PR[GP1:90,2] + 81.361;
   1:L PR[91] 10mm/sec FINE;
   1:  PR[GP1:91,1] = PR[GP1:90,1] + 113.159;
   1:  PR[GP1:91,2] = PR[GP1:90,2] + 81.519;
   1:L PR[91] 10mm/sec FINE;
   1:  PR[GP1:91,1] = PR[GP1:90,1] + 115.962;
   1:  PR[GP1:91,2] = PR[GP1:90,2] + 82.086;
   1:L PR[91] 10mm/sec FINE;
   1:  PR[GP1:91,1] = PR[GP1:90,1] + 118.659;
   1:  PR[GP1:91,2] = PR[GP1:90,2] + 83.080;
   1:L PR[91] 10mm/sec FINE;
   1:  PR[GP1:91,1] = PR[GP1:90,1] + 119.388;
   1:  PR[GP1:91,2] = PR[GP1:90,2] + 83.508;
   1:L PR[91] 10mm/sec FINE;
   1:  PR[GP1:91,1] = PR[GP1:90,1] + 120.774;
   1:  PR[GP1:91,2] = PR[GP1:90,2] + 84.277;
   1:L PR[91] 10mm/sec FINE;
   1:  PR[GP1:91,1] = PR[GP1:90,1] + 121.266;
   1:  PR[GP1:91,2] = PR[GP1:90,2] + 84.569;
   1:L PR[91] 10mm/sec FINE;
   1:  PR[GP1:91,1] = PR[GP1:90,1] + 122.047;
   1:  PR[GP1:91,2] = PR[GP1:90,2] + 85.202;
   1:L PR[91] 10mm/sec FINE;
   1:  PR[GP1:91,1] = PR[GP1:90,1] + 123.234;
   1:  PR[GP1:91,2] = PR[GP1:90,2] + 86.210;
   1:L PR[91] 10mm/sec FINE;
   1:  PR[GP1:91,1] = PR[GP1:90,1] + 124.147;
   1:  PR[GP1:91,2] = PR[GP1:90,2] + 87.214;
   1:L PR[91] 10mm/sec FINE;
   1:  PR[GP1:91,1] = PR[GP1:90,1] + 124.709;
   1:  PR[GP1:91,2] = PR[GP1:90,2] + 87.943;
   1:L PR[91] 10mm/sec FINE;
   1:  PR[GP1:91,1] = PR[GP1:90,1] + 125.445;
   1:  PR[GP1:91,2] = PR[GP1:90,2] + 89.020;
   1:L PR[91] 10mm/sec FINE;
   1:  PR[GP1:91,1] = PR[GP1:90,1] + 125.847;
   1:  PR[GP1:91,2] = PR[GP1:90,2] + 89.853;
   1:L PR[91] 10mm/sec FINE;
   1:  PR[GP1:91,1] = PR[GP1:90,1] + 126.383;
   1:  PR[GP1:91,2] = PR[GP1:90,2] + 90.891;
   1:L PR[91] 10mm/sec FINE;
   1:  PR[GP1:91,1] = PR[GP1:90,1] + 126.731;
   1:  PR[GP1:91,2] = PR[GP1:90,2] + 91.774;
   1:L PR[91] 10mm/sec FINE;
   1:  PR[GP1:91,1] = PR[GP1:90,1] + 127.364;
   1:  PR[GP1:91,2] = PR[GP1:90,2] + 94.158;
   1:L PR[91] 10mm/sec FINE;
   1:  PR[GP1:91,1] = PR[GP1:90,1] + 127.423;
   1:  PR[GP1:91,2] = PR[GP1:90,2] + 94.437;
   1:L PR[91] 10mm/sec FINE;
   1:  PR[GP1:91,1] = PR[GP1:90,1] + 127.495;
   1:  PR[GP1:91,2] = PR[GP1:90,2] + 95.427;
   1:L PR[91] 10mm/sec FINE;
   1:  PR[GP1:91,1] = PR[GP1:90,1] + 127.684;
   1:  PR[GP1:91,2] = PR[GP1:90,2] + 97.477;
   1:L PR[91] 10mm/sec FINE;
   1:  PR[GP1:91,1] = PR[GP1:90,1] + 127.383;
   1:  PR[GP1:91,2] = PR[GP1:90,2] + 100.488;
   1:L PR[91] 10mm/sec FINE;
   1:  PR[GP1:91,1] = PR[GP1:90,1] + 126.865;
   1:  PR[GP1:91,2] = PR[GP1:90,2] + 102.442;
   1:L PR[91] 10mm/sec FINE;
   1:  PR[GP1:91,1] = PR[GP1:90,1] + 126.391;
   1:  PR[GP1:91,2] = PR[GP1:90,2] + 104.412;
   1:L PR[91] 10mm/sec FINE;
   1:  PR[GP1:91,1] = PR[GP1:90,1] + 125.695;
   1:  PR[GP1:91,2] = PR[GP1:90,2] + 105.974;
   1:L PR[91] 10mm/sec FINE;
   1:  PR[GP1:91,1] = PR[GP1:90,1] + 124.777;
   1:  PR[GP1:91,2] = PR[GP1:90,2] + 108.202;
   1:L PR[91] 10mm/sec FINE;
   1:  PR[GP1:91,1] = PR[GP1:90,1] + 123.055;
   1:  PR[GP1:91,2] = PR[GP1:90,2] + 110.842;
   1:L PR[91] 10mm/sec FINE;
   1:  PR[GP1:91,1] = PR[GP1:90,1] + 122.508;
   1:  PR[GP1:91,2] = PR[GP1:90,2] + 111.728;
   1:L PR[91] 10mm/sec FINE;
   1:  PR[GP1:91,1] = PR[GP1:90,1] + 120.974;
   1:  PR[GP1:91,2] = PR[GP1:90,2] + 113.455;
   1:L PR[91] 10mm/sec FINE;
   1:  PR[GP1:91,1] = PR[GP1:90,1] + 119.740;
   1:  PR[GP1:91,2] = PR[GP1:90,2] + 114.815;
   1:L PR[91] 10mm/sec FINE;
   1:  PR[GP1:91,1] = PR[GP1:90,1] + 116.550;
   1:  PR[GP1:91,2] = PR[GP1:90,2] + 117.303;
   1:L PR[91] 10mm/sec FINE;
   1:  PR[GP1:91,1] = PR[GP1:90,1] + 113.153;
   1:  PR[GP1:91,2] = PR[GP1:90,2] + 119.105;
   1:L PR[91] 10mm/sec FINE;
   1:  PR[GP1:91,1] = PR[GP1:90,1] + 109.551;
   1:  PR[GP1:91,2] = PR[GP1:90,2] + 120.206;
   1:L PR[91] 10mm/sec FINE;
   1:  PR[GP1:91,1] = PR[GP1:90,1] + 105.989;
   1:  PR[GP1:91,2] = PR[GP1:90,2] + 120.558;
   1:L PR[91] 10mm/sec FINE;
   1:  PR[GP1:91,1] = PR[GP1:90,1] + 104.980;
   1:  PR[GP1:91,2] = PR[GP1:90,2] + 120.487;
   1:L PR[91] 10mm/sec FINE;
   1:  PR[GP1:91,1] = PR[GP1:90,1] + 104.174;
   1:  PR[GP1:91,2] = PR[GP1:90,2] + 120.410;
   1:L PR[91] 10mm/sec FINE;
   1:  PR[GP1:91,1] = PR[GP1:90,1] + 102.196;
   1:  PR[GP1:91,2] = PR[GP1:90,2] + 120.190;
   1:L PR[91] 10mm/sec FINE;
   1:  PR[GP1:91,1] = PR[GP1:90,1] + 101.481;
   1:  PR[GP1:91,2] = PR[GP1:90,2] + 120.157;
   1:L PR[91] 10mm/sec FINE;
   1:  PR[GP1:91,1] = PR[GP1:90,1] + 97.731;
   1:  PR[GP1:91,2] = PR[GP1:90,2] + 120.175;
   1:L PR[91] 10mm/sec FINE;
   1:  PR[GP1:91,1] = PR[GP1:90,1] + 96.447;
   1:  PR[GP1:91,2] = PR[GP1:90,2] + 120.211;
   1:L PR[91] 10mm/sec FINE;
   1:  PR[GP1:91,1] = PR[GP1:90,1] + 94.053;
   1:  PR[GP1:91,2] = PR[GP1:90,2] + 119.793;
   1:L PR[91] 10mm/sec FINE;
   1:  PR[GP1:91,1] = PR[GP1:90,1] + 92.008;
   1:  PR[GP1:91,2] = PR[GP1:90,2] + 119.495;
   1:L PR[91] 10mm/sec FINE;
   1:  PR[GP1:91,1] = PR[GP1:90,1] + 90.549;
   1:  PR[GP1:91,2] = PR[GP1:90,2] + 118.936;
   1:L PR[91] 10mm/sec FINE;
   1:  PR[GP1:91,1] = PR[GP1:90,1] + 88.012;
   1:  PR[GP1:91,2] = PR[GP1:90,2] + 118.055;
   1:L PR[91] 10mm/sec FINE;
   1:  PR[GP1:91,1] = PR[GP1:90,1] + 87.296;
   1:  PR[GP1:91,2] = PR[GP1:90,2] + 117.584;
   1:L PR[91] 10mm/sec FINE;
   1:  PR[GP1:91,1] = PR[GP1:90,1] + 84.610;
   1:  PR[GP1:91,2] = PR[GP1:90,2] + 115.949;
   1:L PR[91] 10mm/sec FINE;
   1:  PR[GP1:91,1] = PR[GP1:90,1] + 84.391;
   1:  PR[GP1:91,2] = PR[GP1:90,2] + 115.711;
   1:L PR[91] 10mm/sec FINE;
   1:  PR[GP1:91,1] = PR[GP1:90,1] + 81.948;
   1:  PR[GP1:91,2] = PR[GP1:90,2] + 113.243;
   1:L PR[91] 10mm/sec FINE;
   1:  PR[GP1:91,1] = PR[GP1:90,1] + 80.089;
   1:  PR[GP1:91,2] = PR[GP1:90,2] + 109.975;
   1:L PR[91] 10mm/sec FINE;
   1:  PR[GP1:91,1] = PR[GP1:90,1] + 79.119;
   1:  PR[GP1:91,2] = PR[GP1:90,2] + 106.482;
   1:L PR[91] 10mm/sec FINE;
   1:  PR[GP1:91,1] = PR[GP1:90,1] + 79.113;
   1:  PR[GP1:91,2] = PR[GP1:90,2] + 106.425;
   1:L PR[91] 10mm/sec FINE;
   1:  PR[GP1:91,1] = PR[GP1:90,1] + 79.233;
   1:  PR[GP1:91,2] = PR[GP1:90,2] + 102.651;
   1:L PR[91] 10mm/sec FINE;
   1:  PR[GP1:91,1] = PR[GP1:90,1] + 79.355;
   1:  PR[GP1:91,2] = PR[GP1:90,2] + 102.060;
   1:L PR[91] 10mm/sec FINE;
   1:  PR[GP1:91,1] = PR[GP1:90,1] + 80.560;
   1:  PR[GP1:91,2] = PR[GP1:90,2] + 98.194;
   1:L PR[91] 10mm/sec FINE;
   1:  PR[GP1:91,1] = PR[GP1:90,1] + 80.596;
   1:  PR[GP1:91,2] = PR[GP1:90,2] + 98.107;
   1:L PR[91] 10mm/sec FINE;
   1:  PR[GP1:91,1] = PR[GP1:90,1] + 81.070;
   1:  PR[GP1:91,2] = PR[GP1:90,2] + 97.321;
   1:L PR[91] 10mm/sec FINE;
   1:  PR[GP1:91,1] = PR[GP1:90,1] + 82.760;
   1:  PR[GP1:91,2] = PR[GP1:90,2] + 94.326;
   1:L PR[91] 10mm/sec FINE;
   1:  PR[GP1:91,1] = PR[GP1:90,1] + 83.980;
   1:  PR[GP1:91,2] = PR[GP1:90,2] + 93.335;
   1:  PR[GP1:91,3] = PR[GP1:90,3] + 53.900;
   1:L PR[91] 10mm/sec FINE;
   1:  PR[GP1:91,1] = PR[GP1:90,1] + 86.224;
   1:  PR[GP1:91,2] = PR[GP1:90,2] + 90.855;
   1:L PR[91] 10mm/sec FINE;
   1:  PR[GP1:91,1] = PR[GP1:90,1] + 87.908;
   1:  PR[GP1:91,2] = PR[GP1:90,2] + 89.173;
   1:L PR[91] 10mm/sec FINE;
   1:  PR[GP1:91,1] = PR[GP1:90,1] + 89.700;
   1:  PR[GP1:91,2] = PR[GP1:90,2] + 87.826;
   1:L PR[91] 10mm/sec FINE;
   1:  PR[GP1:91,1] = PR[GP1:90,1] + 92.935;
   1:  PR[GP1:91,2] = PR[GP1:90,2] + 85.646;
   1:L PR[91] 10mm/sec FINE;
   1:  PR[GP1:91,1] = PR[GP1:90,1] + 93.696;
   1:  PR[GP1:91,2] = PR[GP1:90,2] + 85.263;
   1:L PR[91] 10mm/sec FINE;
   1:  PR[GP1:91,1] = PR[GP1:90,1] + 96.231;
   1:  PR[GP1:91,2] = PR[GP1:90,2] + 84.158;
   1:L PR[91] 10mm/sec FINE;
   1:  PR[GP1:91,1] = PR[GP1:90,1] + 98.416;
   1:  PR[GP1:91,2] = PR[GP1:90,2] + 83.069;
   1:L PR[91] 10mm/sec FINE;
   1:  PR[GP1:91,1] = PR[GP1:90,1] + 99.276;
   1:  PR[GP1:91,2] = PR[GP1:90,2] + 82.779;
   1:L PR[91] 10mm/sec FINE;
   1:  PR[GP1:91,1] = PR[GP1:90,1] + 103.653;
   1:  PR[GP1:91,2] = PR[GP1:90,2] + 81.498;
   1:L PR[91] 10mm/sec FINE;
   1:  PR[GP1:91,1] = PR[GP1:90,1] + 106.416;
   1:  PR[GP1:91,2] = PR[GP1:90,2] + 81.079;
   1:L PR[91] 10mm/sec FINE;
   1:  PR[GP1:91,1] = PR[GP1:90,1] + 108.785;
   1:  PR[GP1:91,2] = PR[GP1:90,2] + 80.851;
   1:L PR[91] 10mm/sec FINE;
   1:  PR[GP1:91,1] = PR[GP1:90,1] + 108.810;
   1:  PR[GP1:91,2] = PR[GP1:90,2] + 80.865;
   1:L PR[91] 10mm/sec FINE;
   1:  PR[GP1:91,1] = PR[GP1:90,1] + 108.990;
   1:  PR[GP1:91,2] = PR[GP1:90,2] + 80.888;
   1:L PR[91] 10mm/sec FINE;
   1:  PR[GP1:91,1] = PR[GP1:90,1] + 110.540;
   1:  PR[GP1:91,2] = PR[GP1:90,2] + 80.897;
   1:L PR[91] 10mm/sec FINE;
   1:  PR[GP1:91,1] = PR[GP1:90,1] + 112.522;
   1:  PR[GP1:91,2] = PR[GP1:90,2] + 80.968;
   1:L PR[91] 10mm/sec FINE;
   1:  PR[GP1:91,1] = PR[GP1:90,1] + 113.422;
   1:  PR[GP1:91,2] = PR[GP1:90,2] + 81.017;
   1:L PR[91] 10mm/sec FINE;
   1:  PR[GP1:91,1] = PR[GP1:90,1] + 116.294;
   1:  PR[GP1:91,2] = PR[GP1:90,2] + 81.546;
   1:L PR[91] 10mm/sec FINE;
   1:  PR[GP1:91,1] = PR[GP1:90,1] + 117.976;
   1:  PR[GP1:91,2] = PR[GP1:90,2] + 82.128;
   1:L PR[91] 10mm/sec FINE;
   1:  PR[GP1:91,1] = PR[GP1:90,1] + 118.650;
   1:  PR[GP1:91,2] = PR[GP1:90,2] + 82.327;
   1:L PR[91] 10mm/sec FINE;
   1:  PR[GP1:91,1] = PR[GP1:90,1] + 119.843;
   1:  PR[GP1:91,2] = PR[GP1:90,2] + 82.851;
   1:L PR[91] 10mm/sec FINE;
   1:  PR[GP1:91,1] = PR[GP1:90,1] + 121.927;
   1:  PR[GP1:91,2] = PR[GP1:90,2] + 84.052;
   1:L PR[91] 10mm/sec FINE;
   1:  PR[GP1:91,1] = PR[GP1:90,1] + 123.775;
   1:  PR[GP1:91,2] = PR[GP1:90,2] + 85.468;
   1:L PR[91] 10mm/sec FINE;
   1:  PR[GP1:91,1] = PR[GP1:90,1] + 125.277;
   1:  PR[GP1:91,2] = PR[GP1:90,2] + 87.054;
   1:L PR[91] 10mm/sec FINE;
   1:  PR[GP1:91,1] = PR[GP1:90,1] + 126.270;
   1:  PR[GP1:91,2] = PR[GP1:90,2] + 88.480;
   1:L PR[91] 10mm/sec FINE;
   1:  PR[GP1:91,1] = PR[GP1:90,1] + 126.382;
   1:  PR[GP1:91,2] = PR[GP1:90,2] + 88.665;
   1:L PR[91] 10mm/sec FINE;
   1:  PR[GP1:91,1] = PR[GP1:90,1] + 127.080;
   1:  PR[GP1:91,2] = PR[GP1:90,2] + 90.034;
